    30:
        // 5. ASSERT - Weryfikacja końcowa
        AssertTrue(Condition := Cylinder_RetractHappy.Retracted, 
                   Message := 'Cylinder nie zglosil Retracted po powrocie!');
                   
        TEST_FINISHED();
END_CASE
END_METHOD

END_FUNCTION_BLOCK

// ---- POUs/TESTS/FB_ExecutorNCITable_Test.TcPOU
FUNCTION_BLOCK FB_ExecutorNCITable_Test EXTENDS TcUnit.FB_TestSuite
VAR
    Executor         : FB_Exec_Tangential_FeedTable;
    MockChannel      : FB_MockNciChannelFeedTable;

    Executor_Err     : FB_Exec_Tangential_FeedTable;
    MockChannel_Err  : FB_MockNciChannelFeedTable;

    MockProvider     : FB_MockConfigProvider;
    MockAxisX        : FB_MockAxis;
    MockAxisY        : FB_MockAxis;
    MockAxisZ        : FB_MockAxis;
    RecipeBuilder    : FB_PTPRectangle;
END_VAR

Test_Sequence_ExecutesTableCorrectly();
Test_ChannelError_AbortsSequence();

METHOD Test_ChannelError_AbortsSequence
VAR_INST
    Step : INT := 0;
    TimeoutTimer : TON;
END_VAR
TEST('Test_ChannelError_AbortsSequence');

Executor_Err.CyclicLogic();

TimeoutTimer(IN := (Step > 0 AND Step < 100), PT := T#2S);
IF TimeoutTimer.Q THEN
    AssertTrue(FALSE, 'Timeout! Maszyna stanow utknela.');
    TEST_FINISHED();
    Step := 100;
END_IF

CASE Step OF
    0:
        Executor_Err.RecipeBuilder  := RecipeBuilder;
        Executor_Err.ConfigProvider := MockProvider;
        Executor_Err.AxisX          := MockAxisX;
        Executor_Err.AxisY          := MockAxisY;
        Executor_Err.AxisZ          := MockAxisZ;
        Executor_Err.NciChannel     := MockChannel_Err;

        MockAxisX.MockInPosition := TRUE;
        MockAxisY.MockInPosition := TRUE;
        MockAxisZ.MockInPosition := TRUE;
        MockChannel_Err.MockChannelError := FALSE;

        Executor_Err.Execute();
        Step := 10;

    10:
        IF MockChannel_Err.BuildGroupCallCount > 0 THEN
            MockChannel_Err.MockChannelError := TRUE;
            MockChannel_Err.MockChannelErrorId := 4321;
            Step := 20;
        END_IF

    20:
        IF Executor_Err.Error THEN
            AssertEquals_UDINT(Expected := 4321, 
                               Actual := Executor_Err.ErrorID, 
                               Message := 'Executor nie przepisal ErrorID z kanalu tabelarycznego!');
            TEST_FINISHED();
            Step := 100;
        ELSIF Executor_Err.Done THEN
            AssertTrue(Condition := FALSE, Message := 'Executor zignorowal blad kanalu!');
            TEST_FINISHED();
            Step := 100;
        END_IF
END_CASE
END_METHOD

METHOD Test_Sequence_ExecutesTableCorrectly
VAR_INST
    Step         : INT := 0;
    RecipeConfig : ST_RecipeBuilder_Config;
    TimeoutTimer : TON;
END_VAR
TEST('Test_Sequence_ExecutesTableCorrectly');

Executor.CyclicLogic();

TimeoutTimer(IN := (Step > 0 AND Step < 100), PT := T#2S);
IF TimeoutTimer.Q THEN
    AssertTrue(FALSE, 'Timeout! Maszyna stanow utknela.');
    TEST_FINISHED();
    Step := 100;
END_IF

CASE Step OF
    0:
        RecipeConfig.PanelFrontLength := 1000.0;
        RecipeConfig.PanelFrontWidth  := 1000.0; // <- Wymagane, zeby nie ustawilo 0 sztuk!
        RecipeBuilder.Config := RecipeConfig;
        RecipeBuilder.Build();

        Executor.RecipeBuilder  := RecipeBuilder;
        Executor.ConfigProvider := MockProvider;
        Executor.AxisX          := MockAxisX;
        Executor.AxisY          := MockAxisY;
        Executor.AxisZ          := MockAxisZ;
        Executor.NciChannel     := MockChannel; 

        Step := 10;

    10:
        Executor.Execute();
        Step := 20;

    20:
        IF Executor.Busy THEN
            MockAxisX.MockInPosition := TRUE;
            MockAxisY.MockInPosition := TRUE;
            MockAxisZ.MockInPosition := TRUE;
            Step := 30;
        END_IF

    30:
        IF MockChannel.BuildGroupCallCount > 0 THEN
            MockChannel.MockIsGrouped := TRUE; 
            Step := 40;
        END_IF

    40:
        IF MockChannel.StartFeedTableCallCount > 0 THEN
            MockChannel.MockIsFeedingDone := TRUE;
            Step := 50;
        END_IF

    50:
        IF MockChannel.MockIsFeedingDone THEN
            MockChannel.MockIsChannelDone := TRUE;
            Step := 60;
        END_IF

    60:
        IF MockChannel.UngroupCallCount > 0 THEN
            MockChannel.MockIsGrouped := FALSE;
            Step := 70;
        END_IF

    70:
        IF Executor.Done THEN
            AssertTrue(Condition := TRUE, Message := 'Test OK');
            TEST_FINISHED();
            Step := 100;
        ELSIF Executor.Error THEN
            AssertTrue(Condition := FALSE, Message := 'Wystapil nieoczekiwany Error!');
            TEST_FINISHED();
            Step := 100;
        END_IF
END_CASE
END_METHOD

END_FUNCTION_BLOCK

// ---- POUs/TESTS/Mocks/FB_MockNciChannelFeedTable.TcPOU
FUNCTION_BLOCK FB_MockNciChannelFeedTable EXTENDS FB_ComponentBase IMPLEMENTS I_NciChannel_FeedTable
VAR_INPUT
    MockIsGrouped      : BOOL;
    MockIsReady        : BOOL;
    MockChannelError   : BOOL;
    MockChannelErrorId : UDINT;
    MockIsFeedingDone  : BOOL;
    MockIsChannelDone  : BOOL;
END_VAR
VAR_OUTPUT
    BuildGroupCallCount     : INT;
    StartFeedTableCallCount : INT;
    StopCallCount           : INT;
    UngroupCallCount        : INT;
    ResetCallCount          : INT;
END_VAR

METHOD BuildGroup
BuildGroupCallCount := BuildGroupCallCount + 1;
END_METHOD

PROPERTY ChannelError : BOOL
GET
ChannelError := MockChannelError;
END_GET
END_PROPERTY

PROPERTY ChannelErrorId : UDINT
GET
ChannelErrorId := MockChannelErrorId;
END_GET
END_PROPERTY

PROPERTY IsChannelDone : BOOL
GET
IsChannelDone := MockIsChannelDone;
END_GET
END_PROPERTY

PROPERTY IsFeedingDone : BOOL
GET
IsFeedingDone := MockIsFeedingDone;
END_GET
END_PROPERTY

PROPERTY IsGrouped : BOOL
GET
IsGrouped := MockIsGrouped;
END_GET
END_PROPERTY

PROPERTY IsReady : BOOL
GET
IsReady := MockIsReady;
END_GET
END_PROPERTY

METHOD ResetChannel
ResetCallCount := ResetCallCount + 1;
MockChannelError := FALSE;
MockChannelErrorId := 0;
END_METHOD

METHOD StartFeedTable
VAR_IN_OUT
    stTable : ST_NciFeedGroupTable;
END_VAR
StartFeedTableCallCount := StartFeedTableCallCount + 1;
END_METHOD

METHOD Stop
StopCallCount := StopCallCount + 1;
END_METHOD

METHOD Ungroup
UngroupCallCount := UngroupCallCount + 1;
END_METHOD

END_FUNCTION_BLOCK

// ---- POUs/TESTS/Mocks/FB_MockConfigProvider.TcPOU
FUNCTION_BLOCK FB_MockConfigProvider IMPLEMENTS I_GantryConfigProvider
VAR
    _MockConfig : ST_GantryXYZ_Config;
END_VAR

PROPERTY Config : ST_GantryXYZ_Config
GET
Config := _MockConfig;
END_GET
SET
_MockConfig := Config;
END_SET
END_PROPERTY

END_FUNCTION_BLOCK

// ---- POUs/TESTS/Mocks/FB_MockAxis.TcPOU
FUNCTION_BLOCK FB_MockAxis EXTENDS SPT_Components.FB_Component_BasicAxis
VAR
	_Enabled		: BOOL := FALSE;
	
	_MockVelocity     : LREAL;
    _MockAcceleration : LREAL;
    _MockDeceleration : LREAL;
	
	_ForceError	:	BOOL;
END_VAR

VAR_INPUT
    MockInPosition : BOOL := TRUE;
    MockBusy       : BOOL := FALSE;
END_VAR

PROPERTY Acceleration : LREAL
GET
Acceleration := _MockAcceleration;
END_GET
SET
_MockAcceleration := Acceleration;
END_SET
END_PROPERTY

PROPERTY Busy : BOOL
GET
Busy := MockBusy;
END_GET
END_PROPERTY

METHOD CyclicLogic
SUPER^.CyclicLogic();
END_METHOD

PROPERTY Deceleration : LREAL
GET
Deceleration := _MockDeceleration;
END_GET
SET
_MockDeceleration := Deceleration;
END_SET
END_PROPERTY

METHOD Enable : BOOL
SUPER^.Enable(); 
_Enabled := TRUE;
Enable := TRUE;
END_METHOD

PROPERTY Enabled : BOOL
GET
Enabled := _Enabled;
END_GET
END_PROPERTY

PROPERTY Error : BOOL
GET
Error := _Error;
END_GET
END_PROPERTY

PROPERTY ForceError : BOOL
GET
ForceError := _Error;
END_GET
SET
_Error := ForceError;
END_SET
END_PROPERTY

PROPERTY InPosition : BOOL
GET
InPosition := MockInPosition;
END_GET
END_PROPERTY

METHOD MoveAbsolute : BOOL
VAR_INPUT
	Position	  : LREAL;
	AbortPrevious : BOOL;
END_VAR
MockBusy := FALSE;
MockInPosition := TRUE;
END_METHOD

PROPERTY Velocity : LREAL
GET
Velocity := _MockVelocity;
END_GET
SET
_MockVelocity := Velocity;
END_SET
END_PROPERTY

END_FUNCTION_BLOCK

// ---- POUs/TESTS/FB_ExecutorGCode_Test.TcPOU
FUNCTION_BLOCK FB_ExecutorGCode_Test EXTENDS TcUnit.FB_TestSuite
VAR
    Executor         : FB_Exec_Spindle_GCodeXYZ;
    MockChannel      : FB_MockNciChannel;

    Executor_Err     : FB_Exec_Spindle_GCodeXYZ;
    MockChannel_Err  : FB_MockNciChannel;

    MockProvider     : FB_MockConfigProvider;
    MockAxisX        : FB_MockAxis;
    MockAxisY        : FB_MockAxis;
    MockAxisZ        : FB_MockAxis;
    RecipeBuilder    : FB_PTPRectangle;
END_VAR

Test_Sequence_CallsChannelMethodsCorrectly();
Test_ChannelError_AbortsSequence();

METHOD Test_ChannelError_AbortsSequence
VAR_INST
    Step : INT := 0;
    TimeoutTimer : TON;
END_VAR
TEST('Test_ChannelError_AbortsSequence');

Executor_Err.CyclicLogic();

TimeoutTimer(IN := (Step > 0 AND Step < 100), PT := T#2S);
IF TimeoutTimer.Q THEN
    AssertTrue(FALSE, 'Timeout! Maszyna stanow utknela.');
    TEST_FINISHED();
    Step := 100;
END_IF

CASE Step OF
    0:
        Executor_Err.RecipeBuilder  := RecipeBuilder;
        Executor_Err.ConfigProvider := MockProvider;
        Executor_Err.AxisX          := MockAxisX;
        Executor_Err.AxisY          := MockAxisY;
        Executor_Err.AxisZ          := MockAxisZ;
        Executor_Err.NciChannel     := MockChannel_Err;

        MockAxisX.MockInPosition := TRUE;
        MockAxisY.MockInPosition := TRUE;
        MockAxisZ.MockInPosition := TRUE;
        MockChannel_Err.MockChannelError := FALSE;

        Executor_Err.Execute();
        Step := 10;
        
    10:
        IF MockChannel_Err.BuildGroupCallCount > 0 THEN
            MockChannel_Err.MockChannelError := TRUE;
            MockChannel_Err.MockChannelErrorId := 1234;
            Step := 20;
        END_IF

    20:
        IF Executor_Err.Error THEN
            AssertEquals_UDINT(Expected := 1234, 
                               Actual := Executor_Err.ErrorID, 
                               Message := 'Executor nie przepisal ErrorID z kanalu!');
            TEST_FINISHED();
            Step := 100; 
        ELSIF Executor_Err.Done THEN
            AssertTrue(Condition := FALSE, Message := 'Executor zignorowal blad kanalu!');
            TEST_FINISHED();
            Step := 100; 
        END_IF
END_CASE
END_METHOD

METHOD Test_Sequence_CallsChannelMethodsCorrectly
VAR_INST
    Step         : INT := 0;
    RecipeConfig : ST_RecipeBuilder_Config;
    TimeoutTimer : TON;
END_VAR
TEST('Test_Sequence_CallsChannelMethodsCorrectly');

Executor.CyclicLogic();

TimeoutTimer(IN := (Step > 0 AND Step < 100), PT := T#2S);
IF TimeoutTimer.Q THEN
    AssertTrue(FALSE, 'Timeout! Maszyna stanow utknela.');
    TEST_FINISHED();
    Step := 100;
END_IF

CASE Step OF
    0:
        RecipeConfig.PanelFrontLength := 1000.0;
        RecipeConfig.PanelFrontWidth  := 1000.0; // <- Wymagane, zeby nie ustawilo 0 sztuk!
        RecipeBuilder.Config := RecipeConfig;
        RecipeBuilder.Build();

        Executor.RecipeBuilder  := RecipeBuilder;
        Executor.ConfigProvider := MockProvider;
        Executor.AxisX          := MockAxisX;
        Executor.AxisY          := MockAxisY;
        Executor.AxisZ          := MockAxisZ;
        Executor.NciChannel     := MockChannel;
        Step := 10;

    10:
        Executor.Execute();
        Step := 20;

    20:
        IF Executor.Busy THEN
            MockAxisX.MockInPosition := TRUE;
            MockAxisY.MockInPosition := TRUE;
            MockAxisZ.MockInPosition := TRUE;
            Step := 30;
        END_IF

    30:
        IF MockChannel.BuildGroupCallCount > 0 THEN
            MockChannel.MockIsGrouped := TRUE;
            Step := 40;
        END_IF

    40:
        IF MockChannel.LoadProgramCallCount > 0 THEN
            AssertEquals_STRING(Expected := '', Actual := MockChannel.LoadedProgramPath, Message := 'Zla sciezka przekazana do kanalu!');
            MockChannel.MockIsProgramLoaded := TRUE;
            Step := 50;
        END_IF

    50:
        IF MockChannel.StartCallCount > 0 THEN
            MockChannel.MockIsReady := TRUE;
            Step := 60;
        END_IF

    60:
        IF MockChannel.UngroupCallCount > 0 THEN
            MockChannel.MockIsGrouped := FALSE;
            Step := 70;
        END_IF

    70:
        IF Executor.Done THEN
            AssertTrue(Condition := TRUE, Message := 'Test OK');
            TEST_FINISHED();
            Step := 100;
        ELSIF Executor.Error THEN
            AssertTrue(Condition := FALSE, Message := 'Wystapil Error!');
            TEST_FINISHED();
            Step := 100;
        END_IF
END_CASE
END_METHOD

END_FUNCTION_BLOCK

// ---- POUs/TESTS/Mocks/FB_MockNciChannel.TcPOU
FUNCTION_BLOCK FB_MockNciChannel EXTENDS FB_ComponentBase IMPLEMENTS I_NciChannel_GCode
VAR_INPUT
    MockIsGrouped      : BOOL;
    MockIsProgramLoaded: BOOL;
    MockIsReady        : BOOL;
    MockIsMoving       : BOOL;
    MockChannelError   : BOOL;
    MockChannelErrorId : UDINT;
END_VAR
VAR_OUTPUT
    BuildGroupCallCount : INT;
    LoadProgramCallCount: INT;
    StartCallCount      : INT;
    StopCallCount       : INT;
    UngroupCallCount    : INT;
    ResetCallCount      : INT;
    LoadedProgramPath   : STRING(255);
END_VAR

METHOD BuildGroup
BuildGroupCallCount := BuildGroupCallCount + 1;
END_METHOD

PROPERTY ChannelError : BOOL
GET
ChannelError := MockChannelError;
END_GET
END_PROPERTY

PROPERTY ChannelErrorId : UDINT
GET
ChannelErrorId := MockChannelErrorId;
END_GET
END_PROPERTY

PROPERTY IsGrouped : BOOL
GET
IsGrouped := MockIsGrouped;
END_GET
END_PROPERTY

PROPERTY IsMoving : BOOL
GET
IsMoving := MockIsMoving;
END_GET
END_PROPERTY

PROPERTY IsProgramLoaded : BOOL
GET
IsProgramLoaded := MockIsProgramLoaded;
END_GET
END_PROPERTY

PROPERTY IsReady : BOOL
GET
IsReady := MockIsReady;
END_GET
END_PROPERTY

METHOD LoadProgram
VAR_INPUT
    sProgramPath : STRING(255);
END_VAR
LoadProgramCallCount := LoadProgramCallCount + 1;
LoadedProgramPath := sProgramPath;
END_METHOD

METHOD ResetChannel
ResetCallCount := ResetCallCount + 1;
MockChannelError := FALSE;
MockChannelErrorId := 0;
END_METHOD

METHOD Start
StartCallCount := StartCallCount + 1;
END_METHOD

METHOD Stop
StopCallCount := StopCallCount + 1;
END_METHOD

METHOD Ungroup
UngroupCallCount := UngroupCallCount + 1;
END_METHOD

END_FUNCTION_BLOCK

// ---- POUs/TESTS/FB_FeedBuilderRoundedRect_Test.TcPOU
FUNCTION_BLOCK FB_FeedBuilderRoundedRect_Test EXTENDS TcUnit.FB_TestSuite
VAR
    Builder    : FB_FeedRoundedRectangle;
    MockWriter : FB_MockGeometryWriter;
    Config     : ST_RecipeBuilder_Config;
END_VAR

Test_Calculates_Footprint_And_StartPoint();
Test_Generates_Lines_And_Arcs_With_Radius();
Test_Zero_Radius_Generates_Only_Lines();

METHOD Test_Calculates_Footprint_And_StartPoint
VAR
    WasBuilt : BOOL;
END_VAR
TEST('Test_Calculates_Footprint_And_StartPoint');

// 1. ARRANGE
Config.PanelFrontWidth  := 300.0;
Config.PanelFrontLength := 400.0;
Config.Radius           := 10.0;
Config.CuttingOverpass  := 0.0; // Upraszczamy Footprint
Config.GroovingOverpass := 0.0;

Builder.Config := Config;
Builder.GeometryWriter := MockWriter; // Wstrzykujemy mock

// 2. ACT
WasBuilt := Builder.Build();

// 3. ASSERT
AssertTrue(Condition := WasBuilt, Message := 'Recepta zwrocila FALSE przy probie Build()!');

AssertEquals_REAL(Expected := 300.0, 
                  Actual := Builder.FootprintX, 
                  Delta := 0.01, 
                  Message := 'Zle wyliczony FootprintX dla zaokraglonego prostokata!');

AssertEquals_REAL(Expected := 400.0, 
                  Actual := Builder.FootprintY, 
                  Delta := 0.01, 
                  Message := 'Zle wyliczony FootprintY dla zaokraglonego prostokata!');

// Sprawdzamy czy start w osi X to srodek detalu (zgodnie z kodem TotalX / 2.0)
AssertEquals_LREAL(Expected := 150.0, 
                   Actual := MockWriter.LastStartX, 
                   Delta := 0.01, 
                   Message := 'Punt Startowy NCI X nie znajduje sie na srodku dolnej krawedzi!');

TEST_FINISHED();
END_METHOD

METHOD Test_Generates_Lines_And_Arcs_With_Radius
VAR
    WasBuilt : BOOL;
END_VAR
TEST('Test_Generates_Lines_And_Arcs_With_Radius');

// 1. ARRANGE
Config.PanelFrontWidth  := 200.0;
Config.PanelFrontLength := 300.0;
Config.Radius           := 20.0;
Builder.Config := Config;
Builder.GeometryWriter := MockWriter;

// Uzywamy nowej metody do resetowania mocka
MockWriter.ResetCounters();

// 2. ACT
WasBuilt := Builder.Build();

// 3. ASSERT
// 4 rogi z promieniem > 0 powinny wygenerować 4 łuki
AssertEquals_INT(Expected := 4, 
                 Actual := MockWriter.AddArcCount, 
                 Message := 'Oczekiwano wygenerowania 4 lukow (AddArc)!');

// Dojazd od punktu srodkowego (1), miedzy 4 rogami (3), i powrot do srodka (1) = 5 linii.
AssertEquals_INT(Expected := 5, 
                 Actual := MockWriter.AddLineCount, 
                 Message := 'Oczekiwano wygenerowania 5 linii prostych (AddLine)!');

TEST_FINISHED();
END_METHOD

METHOD Test_Zero_Radius_Generates_Only_Lines
VAR
    WasBuilt : BOOL;
END_VAR
TEST('Test_Zero_Radius_Generates_Only_Lines');

// 1. ARRANGE
Config.PanelFrontWidth  := 200.0;
Config.PanelFrontLength := 300.0;
Config.Radius           := 0.0; // Promień ZERO (ostry prostokąt)
Builder.Config := Config;
Builder.GeometryWriter := MockWriter;

// Uzywamy nowej metody do resetowania mocka
MockWriter.ResetCounters();

// 2. ACT
WasBuilt := Builder.Build();

// 3. ASSERT
// Przy promieniu = 0 kod recepty ma warunek IF Radius > 0, wiec łuki się nie dodadzą
AssertEquals_INT(Expected := 0, 
                 Actual := MockWriter.AddArcCount, 
                 Message := 'Przy promieniu 0 wygenerowano luki!');

AssertEquals_INT(Expected := 5, 
                 Actual := MockWriter.AddLineCount, 
                 Message := 'Oczekiwano wygenerowania 5 linii prostych (prostokat bez zaokraglen)!');

TEST_FINISHED();
END_METHOD

END_FUNCTION_BLOCK

// ---- POUs/TESTS/Mocks/FB_MockGeometryWriter.TcPOU
FUNCTION_BLOCK FB_MockGeometryWriter IMPLEMENTS I_GeometryWriter
VAR_OUTPUT
    ClearCount                     : INT;
    EnableTangentialFollowingCount : INT;
    AddStartPointCount             : INT;
    AddLineCount                   : INT;
    AddArcCount                    : INT;
    EndTableCount                  : INT;
    
    // Ostatnie parametry ze StartPoint (do weryfikacji)
    LastStartX : LREAL;
    LastStartY : LREAL;
END_VAR

METHOD AddArc : BOOL
VAR_INPUT
    TargetX    : LREAL;
    TargetY    : LREAL;
    CenterX    : LREAL;
    CenterY    : LREAL;
    Velo       : LREAL;
    Clockwise  : BOOL;
END_VAR
AddArcCount := AddArcCount + 1;
AddArc := TRUE;
END_METHOD

METHOD AddLine : BOOL
VAR_INPUT
    TargetX : LREAL;
    TargetY : LREAL;
    Velo    : LREAL;
END_VAR
AddLineCount := AddLineCount + 1;
AddLine := TRUE;
END_METHOD

METHOD AddStartPoint : BOOL
VAR_INPUT
    TargetX : LREAL;
    TargetY : LREAL;
END_VAR
AddStartPointCount := AddStartPointCount + 1;
LastStartX := TargetX;
LastStartY := TargetY;
AddStartPoint := TRUE;
END_METHOD

METHOD Clear : BOOL
VAR_INPUT
END_VAR
ClearCount := ClearCount + 1;
Clear := TRUE;
END_METHOD

METHOD EnableTangentialFollowing : BOOL
VAR_INPUT
END_VAR
EnableTangentialFollowingCount := EnableTangentialFollowingCount + 1;
EnableTangentialFollowing := TRUE;
END_METHOD

METHOD EndTable : BOOL
VAR_INPUT
END_VAR
EndTableCount := EndTableCount + 1;
EndTable := TRUE;
END_METHOD

METHOD ResetCounters
ClearCount := 0;
EnableTangentialFollowingCount := 0;
AddStartPointCount := 0;
AddLineCount := 0;
AddArcCount := 0;
EndTableCount := 0;
LastStartX := 0.0;
LastStartY := 0.0;
END_METHOD

END_FUNCTION_BLOCK

// ---- POUs/TESTS/FB_NciChannelTangential_Test.TcPOU
FUNCTION_BLOCK FB_NciChannelTangential_Test EXTENDS TcUnit.FB_TestSuite
VAR
    ChannelTan  : FB_NciChannelTangential;
    DummyTable  : ST_NciFeedGroupTable;
END_VAR

Test_StartFeedTable_ResetsDoneFlags();
Test_ResetChannel_ClearsErrors();
Test_BuildExtGroup_ClearsGroupedFlag();

METHOD Test_BuildExtGroup_ClearsGroupedFlag
VAR_INST
END_VAR
TEST('Test_BuildExtGroup_ClearsGroupedFlag');

// ACT - Budowanie grupy zawierającej dodatkowo oś Q1
ChannelTan.BuildGroup();

// ASSERT
AssertFalse(Condition := ChannelTan.IsGrouped,
            Message := 'IsGrouped nie zostalo zresetowane przy wywolaniu BuildGroup na EXT grupie!');
AssertFalse(Condition := ChannelTan.ChannelError,
            Message := 'Bledy kanalu tangencjalnego nie zostaly zresetowane przy probie BuildGroup!');

TEST_FINISHED();
END_METHOD

METHOD Test_ResetChannel_ClearsErrors
VAR_INST
END_VAR
TEST('Test_ResetChannel_ClearsErrors');

// ACT
ChannelTan.ResetChannel();

// ASSERT
AssertFalse(Condition := ChannelTan.ChannelError,
            Message := 'Flaga bledu kanalu tangencjalnego nie zniknela po wywolaniu ResetChannel!');
AssertEquals_UDINT(Expected := 0, 
                   Actual := ChannelTan.ChannelErrorId, 
                   Message := 'ID bledu nie zostalo wyzerowane w kanale tangencjalnym!');

TEST_FINISHED();
END_METHOD

METHOD Test_StartFeedTable_ResetsDoneFlags
VAR_INST
END_VAR
TEST('Test_StartFeedTable_ResetsDoneFlags');

// ACT - Przekazujemy strukturę z tabelą i startujemy feedowanie punktów
ChannelTan.StartFeedTable(stTable := DummyTable);

// ASSERT - Flagi końca powinny być natychmiast wyzerowane
AssertFalse(Condition := ChannelTan.IsFeedingDone,
            Message := 'IsFeedingDone powinno byc FALSE na starcie interpolacji tabelarycznej!');
AssertFalse(Condition := ChannelTan.IsChannelDone,
            Message := 'IsChannelDone powinno byc FALSE na starcie interpolacji tabelarycznej!');

TEST_FINISHED();
END_METHOD

END_FUNCTION_BLOCK

// ---- POUs/TESTS/FB_NciChannel_Test.TcPOU
FUNCTION_BLOCK FB_NciChannel_Test EXTENDS TcUnit.FB_TestSuite
VAR
    Channel : FB_NciChannel;
END_VAR

Test_LoadProgram_ClearsLoadedFlag();
Test_ResetChannel_ClearsErrors();
Test_BuildGroup_ClearsGroupedFlag();
Test_Real_BuildGroup_Integration();
Test_DisconnectedState_ReturnsNotReady();

METHOD Test_BuildGroup_ClearsGroupedFlag
VAR_INST
    Executed : BOOL;
END_VAR
TEST('Test_BuildGroup_ClearsGroupedFlag');
IF NOT Executed THEN
    Channel.BuildGroup();
    AssertFalse(Condition := Channel.IsGrouped, Message := 'IsGrouped nie zostalo zresetowane przy wywolaniu BuildGroup!');
    AssertFalse(Condition := Channel.ChannelError, Message := 'Bledy kanalu nie zostaly zresetowane przy probie BuildGroup!');
    TEST_FINISHED();
    Executed := TRUE;
END_IF
END_METHOD

METHOD Test_DisconnectedState_ReturnsNotReady
VAR_INST
    Executed : BOOL;
END_VAR
TEST('Test_DisconnectedState_ReturnsNotReady');
IF NOT Executed THEN
    AssertFalse(Condition := Channel.IsReady, Message := 'IsReady zwrocilo TRUE pomimo braku fizycznego polaczenia z NC!');
    AssertFalse(Condition := Channel.IsMoving, Message := 'IsMoving zwrocilo TRUE pomimo braku fizycznego polaczenia z NC!');
    TEST_FINISHED();
    Executed := TRUE;
END_IF
END_METHOD

METHOD Test_LoadProgram_ClearsLoadedFlag
VAR_INST
    Executed : BOOL;
END_VAR
TEST('Test_LoadProgram_ClearsLoadedFlag');
IF NOT Executed THEN
    Channel.LoadProgram('C:\test_path.nc');
    AssertFalse(Condition := Channel.IsProgramLoaded, Message := 'Flaga IsProgramLoaded nie zostala zresetowana!');
    TEST_FINISHED();
    Executed := TRUE;
END_IF
END_METHOD

METHOD Test_Real_BuildGroup_Integration
VAR_INST
    Step : INT := 0;
    TimeoutTimer : TON;
END_VAR
TEST('Test_Real_BuildGroup_Integration');

// Wstrzykujemy ID osi testowych (odczytane z Twojego tsproj) oraz poprawne ID grupy
Channel.stAxisIds.nX := 5; 
Channel.stAxisIds.nY := 6;
Channel.stAxisIds.nZ := 7;
Channel.nGroupId := 11; // Wirtualna grupa NCI dla testow to 11

Channel.CyclicLogic();

CASE Step OF
    0:
        Channel.BuildGroup();
        Step := 10;

    10:
        TimeoutTimer(IN := TRUE, PT := T#3S);
        
        IF Channel.IsGrouped THEN
            Step := 20;
        ELSIF Channel.ChannelError THEN
            AssertTrue(Condition := FALSE, Message := CONCAT('NC zwrocilo blad! ErrorID: ', UDINT_TO_STRING(Channel.ChannelErrorId)));
            TEST_FINISHED();
        ELSIF TimeoutTimer.Q THEN
            AssertTrue(Condition := FALSE, Message := 'Timeout! NC nie odpowiedzialo.');
            TEST_FINISHED();
        END_IF

    20:
        AssertTrue(Condition := Channel.IsGrouped, Message := 'Grupa powinna byc zgloszona jako gotowa!');
        Channel.Ungroup();
        Step := 30;

    30:
        IF NOT Channel.IsGrouped THEN
            TimeoutTimer(IN := FALSE);
            TEST_FINISHED();
            Step := 100;
        END_IF
END_CASE
END_METHOD

METHOD Test_ResetChannel_ClearsErrors
VAR_INST
    Executed : BOOL;
END_VAR
TEST('Test_ResetChannel_ClearsErrors');
IF NOT Executed THEN
    Channel.ResetChannel();
    AssertFalse(Condition := Channel.ChannelError, Message := 'Flaga bledu kanalu nie zniknela po wywolaniu ResetChannel!');
    AssertEquals_UDINT(Expected := 0, Actual := Channel.ChannelErrorId, Message := 'ID bledu nie zostalo wyzerowane!');
    TEST_FINISHED();
    Executed := TRUE;
END_IF
END_METHOD

END_FUNCTION_BLOCK

// ---- POUs/TESTS/FB_GantryXYZ_Test.TcPOU
FUNCTION_BLOCK FB_GantryXYZ_Test EXTENDS TcUnit.FB_TestSuite
VAR
	Gantry : FB_GantryXYZ;
END_VAR

Test_ApplyProfile_Applies_Correct_Dynamics();
Test_Speeds_Never_Zero_Or_Negative();
//Test_StateChanged_Updates_Profile(); //Needs to be investigated

METHOD Test_ApplyProfile_Applies_Correct_Dynamics
VAR_INPUT
END_VAR
TEST('Test_ApplyProfile_Applies_Correct_Dynamics');

// 1. ACT - Aplikujemy profil Homing (powolny, otwarte limity)
Gantry.ApplyProfile(E_MachineProfile.eHoming);

// 2. ASSERT - Akceleracja osi X powinna wynosić 200.0
AssertEquals_LREAL(Expected := 200.0, 
                   Actual := Gantry.RefAxisX.Acceleration, 
                   Delta := 0.01, 
                   Message := 'ApplyProfile: Blad akceleracji X dla profilu Homing');

// 3. ACT - Aplikujemy profil Production (agresywny)
Gantry.ApplyProfile(E_MachineProfile.eProduction);

// 4. ASSERT - Akceleracja osi X powinna wynosić 1500.0
AssertEquals_LREAL(Expected := 1500.0, 
                   Actual := Gantry.RefAxisX.Acceleration, 
                   Delta := 0.01, 
                   Message := 'ApplyProfile: Blad akceleracji X dla profilu Production');

// 5. ACT - Aplikujemy profil Manual (pośredni)
Gantry.ApplyProfile(E_MachineProfile.eManual);

// 6. ASSERT - Akceleracja osi X powinna wynosić 500.0
AssertEquals_LREAL(Expected := 500.0, 
                   Actual := Gantry.RefAxisX.Acceleration, 
                   Delta := 0.01, 
                   Message := 'ApplyProfile: Blad akceleracji X dla profilu Manual');

TEST_FINISHED();
END_METHOD

METHOD Test_Speeds_Never_Zero_Or_Negative
VAR
    BadConfig    : ST_GantryXYZ_Config;
    ActualConfig : ST_GantryXYZ_Config;
END_VAR
TEST('Test_Speeds_Never_Zero_Or_Negative');

// 1. ARRANGE - Złe dane (np. wpisane przez uszkodzone HMI lub błąd ludzki)
BadConfig.RapidSpeedX := 0.0;        // Zero! Oś nigdy nie dojedzie, zawiesi maszynę stanów
BadConfig.CuttingSpeedXY := -50.0;    // Ujemna prędkość!
BadConfig.GroovingSpeedZ := -0.01;   // Prędkość zagłębiania bliska 0/ujemna
BadConfig.CuttingIdleTime := -2.0;   // Ujemny czas postoju? Timer zwariuje

// 2. ACT - Próba wstrzyknięcia do Gantry
Gantry.Config := BadConfig;
ActualConfig := Gantry.Config; // Odczytujemy stan po "obronie" przez Set

// 3. ASSERT - Sprawdzamy czy Gantry ustawiło bezpieczne minima
AssertEquals_REAL(Expected := 1.0, 
                  Actual := ActualConfig.RapidSpeedX, 
                  Delta := 0.01, 
                  Message := 'RapidSpeedX rowne 0 zostalo przepuszczone!');

AssertEquals_REAL(Expected := 1.0, 
                  Actual := ActualConfig.CuttingSpeedXY, 
                  Delta := 0.01, 
                  Message := 'Ujemna predkosc ciecia przeszla do systemu!');

AssertEquals_REAL(Expected := 1.0, 
                  Actual := ActualConfig.GroovingSpeedZ, 
                  Delta := 0.01, 
                  Message := 'Ujemna/Zerowa predkosc zaglabiania (Z) przeszla!');
                  
AssertEquals_REAL(Expected := 0.0, 
                  Actual := ActualConfig.CuttingIdleTime, 
                  Delta := 0.01, 
                  Message := 'Ujemny czas oczekiwania przeszedl do systemu!');

TEST_FINISHED();
END_METHOD

METHOD Test_StateChanged_Updates_Profile
VAR_INST
    Step : INT := 0;
    Watchdog : TON; // Zabezpieczenie przed zawieszeniem IDE
END_VAR
TEST('Test_StateChanged_Updates_Profile');

// Krytyczne: Wywołujemy logikę Gantry raz na cykl PLC, BEZ ŻADNYCH PĘTLI WHILE/FOR!
Gantry.CyclicLogic();

// Zabezpieczenie testu: jeżeli maszyna PackML utknie i nie zmieni stanu,
// po 2 sekundach przerywamy test, by chronić IDE przed zawieszeniem.
Watchdog(IN := (Step > 0 AND Step < 100), PT := T#2S);
IF Watchdog.Q THEN
    AssertTrue(Condition := FALSE, Message := 'Timeout testu - PackML utknelo w jednym ze stanow! Prawdopodobnie odrzucono komende.');
    TEST_FINISHED();
    Step := 100; // Blokada przed dalszym wykonywaniem
END_IF

CASE Step OF
    0:
        // 1. Zmieniamy tryb na Manualny (od razu na starcie)
        Gantry.ChangeMode(E_PMLUnitMode.ePMLUnitMode_Manual);
        Step := 5;

    5:
        // Czekamy aż PackML fizycznie "zrozumie" zmianę trybu
        IF Gantry.CurrentMode = E_PMLUnitMode.ePMLUnitMode_Manual THEN
            // Zrzucamy maszynę do bezpiecznego stanu Aborted
            Gantry.ChangeState(E_PMLCommand.ePMLCommand_Abort);
            Step := 10;
        END_IF

    10:
        // Czekamy na wejście w Aborted
        IF Gantry.CurrentState = E_PMLState.ePMLState_Aborted THEN
            
            // W trybie Manual zawsze profil ma być ustawiony na Acc=500.0
            AssertEquals_LREAL(Expected := 500.0, 
                               Actual := Gantry.RefAxisX.Acceleration, 
                               Delta := 0.01, 
                               Message := 'Tryb Manualny nie zaladowal prawidlowego profilu!');

            // Zmieniamy tryb z powrotem na produkcyjny
            Gantry.ChangeMode(E_PMLUnitMode.ePMLUnitMode_Production);
            Step := 15;
        END_IF

    15:
        // Czekamy aż PackML potwierdzi tryb produkcyjny
        IF Gantry.CurrentMode = E_PMLUnitMode.ePMLUnitMode_Production THEN
            // Ze stanu Aborted przechodzimy komendą Clear
            Gantry.ChangeState(E_PMLCommand.ePMLCommand_Clear);
            Step := 20;
        END_IF
        
    20:
        // Maszyna po "Clearing" wejdzie w stan "Stopped"
        IF Gantry.CurrentState = E_PMLState.ePMLState_Stopped THEN
            
            // DOPIERO stąd można bezpiecznie wezwać komendę Reset!
            Gantry.ChangeState(E_PMLCommand.ePMLCommand_Reset);
            Step := 30;
        END_IF

    30:
        // Łapiemy moment wejścia w Resetting
        IF Gantry.CurrentState = E_PMLState.ePMLState_Resetting THEN
            
            // To nasz ostateczny sprawdzian: StateChanged() powinno było podmienić profil!
            AssertEquals_LREAL(Expected := 200.0, 
                               Actual := Gantry.RefAxisX.Acceleration, 
                               Delta := 0.01, 
                               Message := 'Rozpoczecie bazowania (Resetting) nie zmienilo profilu maszyny na Homing!');
                               
            TEST_FINISHED(); // Sukces!
            Step := 100; // Koniec
        END_IF
END_CASE
END_METHOD

END_FUNCTION_BLOCK

// ---- POUs/TESTS/FB_ExecutorCut_Test.TcPOU
FUNCTION_BLOCK FB_ExecutorCut_Test EXTENDS TcUnit.FB_TestSuite 
VAR
    Executor : FB_Exec_Pneumatic_PTP;
	Executor_Unhappy     : FB_Exec_Pneumatic_PTP;
	
	MockConfigProvider : FB_MockConfigProvider;

    MockCylinder : FB_MockCylinder;
	MockCylinder_Unhappy : FB_MockCylinder;
    MockAxisX    : FB_MockAxis := (Name := 'MockX');
    MockAxisY    : FB_MockAxis := (Name := 'MockY');
    MockAxisZ    : FB_MockAxis := (Name := 'MockZ');
    
    TestRecipe   : FB_PTPBorgoWings;

	
	Executor_Zero       : FB_Exec_Pneumatic_PTP;
    MockCylinder_Zero   : FB_MockCylinder;
    BuilderArona        : FB_PTPArona; // Arona to nasza wydmuszka, zwraca 0 segmentów!

    Executor_AxisErr    : FB_Exec_Pneumatic_PTP;
    MockAxisX_Err       : FB_MockAxis;

    Executor_CutY       : FB_Exec_Pneumatic_PTP;
    MockCylinder_CutY   : FB_MockCylinder;
	
	Executor_Nesting : FB_Exec_Pneumatic_PTP;
    MockCylinder_Nesting : FB_MockCylinder;
	
END_VAR

Test_AxisError_AbortsSequence();
Test_Executes_CutY_Direction();
Test_Executes_Nesting_Copies();
Test_Sequence_AbortsOnCylinderError();
Test_Sequence_ExecutesCutsCorrectly();
Test_ZeroSegments_FinishesImmediately();

METHOD Test_AxisError_AbortsSequence
VAR_INST
    i : INT;
    RecipeConfig : ST_RecipeBuilder_Config; 
END_VAR


TEST('Test_AxisError_AbortsSequence');

// 1. ARRANGE - Używamy poprawnej receptury (BorgoWings)
RecipeConfig.PanelFrontLength := 1000.0;  
TestRecipe.Config := RecipeConfig;        
TestRecipe.Build();                       
Executor_AxisErr.RecipeBuilder  := TestRecipe; 
Executor_AxisErr.ConfigProvider := MockConfigProvider; // Poprawiona nazwa
Executor_AxisErr.Cylinder       := MockCylinder;
Executor_AxisErr.AxisX          := MockAxisX_Err; // Podpinamy złośliwą oś
Executor_AxisErr.AxisY          := MockAxisY;
Executor_AxisErr.AxisZ          := MockAxisZ;
Executor_AxisErr.CutDirection   := E_CutDirection.eCutX;

MockAxisX_Err.ForceError := TRUE; // Zmuszamy oś do błędu!

// 2. ACT
Executor_AxisErr.Execute();

// Puszczamy maszynę stanów. Wpadnie do kroku 10 (dojazd), potem 20 i od razu zobaczy błąd osi (skok do 999).
FOR i := 1 TO 10 DO
    Executor_AxisErr.CyclicLogic();
END_FOR

// 3. ASSERT
AssertTrue(Condition := Executor_AxisErr.Error, 
           Message := 'Executor nie zglosil bledu, gdy os ulegla awarii!');

AssertFalse(Condition := Executor_AxisErr.Done, 
            Message := 'Executor zglosil sukces (Done), pomimo bledu osi!');

TEST_FINISHED();
END_METHOD

METHOD Test_Executes_CutY_Direction
VAR_INST
    Step : INT := 0;
    RecipeConfig : ST_RecipeBuilder_Config;
END_VAR
TEST('Test_Executes_CutY_Direction');

Executor_CutY.CyclicLogic();

CASE Step OF
    0:
        // 1. ARRANGE - Receptura BorgoWings ma dokładnie 6 cięć Y
        RecipeConfig.PanelFrontLength := 1000.0;
        TestRecipe.Config := RecipeConfig;
        TestRecipe.Build(); 
        
        Executor_CutY.RecipeBuilder  := TestRecipe;
		Executor_CutY.ConfigProvider := MockConfigProvider;
        Executor_CutY.Cylinder       := MockCylinder_CutY;
        Executor_CutY.AxisX          := MockAxisX;
        Executor_CutY.AxisY          := MockAxisY;
        Executor_CutY.AxisZ          := MockAxisZ;
        
        // Ustawiamy cięcie wzdłuż osi Y!
        Executor_CutY.CutDirection   := E_CutDirection.eCutY; 
        
        Step := 10;
        
    10:
        // 2. ACT
        Executor_CutY.Execute();
        Step := 20;
        
    20:
        // Czekamy na koniec asynchronicznej sekwencji
        IF Executor_CutY.Done THEN
            Step := 30;
        ELSIF Executor_CutY.Error THEN
            AssertTrue(FALSE, 'Wyrzucono blad podczas ciecia Y!');
            TEST_FINISHED();
        END_IF
        
    30:
        // 3. ASSERT - Weryfikujemy ilość cięć (BorgoWings = 6)
        AssertEquals_INT(Expected := 6, 
                         Actual := MockCylinder_CutY.ExtendCallCount, 
                         Message := 'Zla liczba wysuniec cylindra przy cieciu Y!');
                         
        TEST_FINISHED();
END_CASE
END_METHOD

METHOD Test_Executes_Nesting_Copies
VAR_INST
    Step         : INT := 0;
    RecipeConfig : ST_RecipeBuilder_Config;
    TestConfig   : ST_GantryXYZ_Config;
    

    LocalTestRecipe : FB_PTPBorgoWings;
    LocalConfigProvider : FB_MockConfigProvider;
END_VAR
TEST('Test_Executes_Nesting_Copies');
Executor_Nesting.CyclicLogic(); 

CASE Step OF
    0:
        // 1. ARRANGE
        // Wykorzystujemy BorgoWings, które domyślnie posiada 6 segmentów CutX
        RecipeConfig.PanelFrontLength := 300.0;
        RecipeConfig.PanelHeight := 100.0;
        RecipeConfig.PanelFrontWidth := 300.0;
        
        // Wymuszamy 2 kopie w X i 2 kopie w Y
        RecipeConfig.FillAll := FALSE;
        RecipeConfig.RequestedCopiesX := 2;
        RecipeConfig.RequestedCopiesY := 2;
        
        LocalTestRecipe.Config := RecipeConfig;
        LocalTestRecipe.Build(); 
        
        TestConfig.CuttingSpeedXY := 100;
        TestConfig.RapidSpeedX := 100;
        TestConfig.CuttingIdleTime := 0.0;
        // Szybki test
        
        // Podpinamy wyizolowane zależności
        LocalConfigProvider.Config := TestConfig;
        Executor_Nesting.RecipeBuilder  := LocalTestRecipe;
        Executor_Nesting.ConfigProvider := LocalConfigProvider;
        Executor_Nesting.Cylinder       := MockCylinder_Nesting;
        Executor_Nesting.AxisX          := MockAxisX;
        Executor_Nesting.AxisY          := MockAxisY;
        Executor_Nesting.AxisZ          := MockAxisZ;
        Executor_Nesting.CutDirection   := E_CutDirection.eCutX; 
        
        Step := 10;
        
    10:
        // 2. ACT
        Executor_Nesting.Execute();
        Step := 20;
        
    20:
        IF Executor_Nesting.Done THEN
            Step := 30;
        ELSIF Executor_Nesting.Error THEN
            AssertTrue(FALSE, 'Executor zwrocil Error zamiast Done przy Nestingu!');
            TEST_FINISHED();
        END_IF
        
    30:
        // 3. ASSERT
        // BorgoWings ma 6 cięć X na jedną sztukę.
        // 2 kopie X * 2 kopie Y = 4 sztuki.
        // 4 sztuki * 6 cięć = 24 wysunięcia siłownika!
        AssertEquals_INT(Expected := 24, 
                         Actual := MockCylinder_Nesting.ExtendCallCount, 
                         Message := 'Zla liczba ciec przy multiplexowaniu (Nestingu)!');
        TEST_FINISHED();
END_CASE
END_METHOD

METHOD Test_Sequence_AbortsOnCylinderError
VAR_INST
    Step : INT := 0;
    RecipeConfig : ST_RecipeBuilder_Config;
	TestConfig : ST_GantryXYZ_Config;
END_VAR


TEST('Test_Sequence_AbortsOnCylinderError');

Executor_Unhappy.CyclicLogic();

CASE Step OF
    0:
        // 1. ARRANGE - Przygotowanie receptury BorgoWings (6 cięć)
        RecipeConfig.PanelFrontLength := 1000.0;
        TestRecipe.Config := RecipeConfig;
        TestRecipe.Build(); 
		
		TestConfig.CuttingSpeedXY := 10;    
		TestConfig.GroovingSpeedXY := 10;
		TestConfig.RapidSpeedX := 10;
		TestConfig.RapidSpeedY := 10;
	
        
        TestConfig.CuttingIdleTime := 0.0; 
        
        // ZMUSZAMY MOCK DO AWARII PRZY 3. PRÓBIE WYSUNIĘCIA
        MockCylinder_Unhappy.FailOnExtendCount := 3;
        
        // Wstrzykujemy zależności do Executora "Unhappy"
		MockConfigProvider.Config := TestConfig; 
		Executor_Unhappy.RecipeBuilder  := TestRecipe;
		Executor_Unhappy.ConfigProvider := MockConfigProvider; 
        Executor_Unhappy.Cylinder       := MockCylinder_Unhappy;
        Executor_Unhappy.AxisX          := MockAxisX;
        Executor_Unhappy.AxisY          := MockAxisY;
        Executor_Unhappy.AxisZ          := MockAxisZ;
        
        Step := 10;
        
    10:
        // 2. ACT - Start maszyny
        Executor_Unhappy.Execute();
        Step := 20;
        
    20:
        // 3. ASSERT - Oczekujemy BŁĘDU, a nie zakończenia sukcesem!
        IF Executor_Unhappy.Error THEN
            Step := 30; // Sukces testu - Executor wyrzucił błąd
        ELSIF Executor_Unhappy.Done THEN
            AssertTrue(FALSE, 'Cylinder zglosil blad, a Executor zignorowal to i zakonczyl sukcesem!');
            TEST_FINISHED();
        END_IF
        
    30:
        // 4. ASSERT - Weryfikacja dokładnego zachowania podczas awarii
        
        // Oczekujemy, że wysunięcie zostało wywołane dokładnie 3 razy i ani razu więcej
        AssertEquals_INT(Expected := 3, 
                         Actual := MockCylinder_Unhappy.ExtendCallCount, 
                         Message := 'Executor nie zatrzymal sie po bledzie na 3. cieciu!');
                         
        // Oczekujemy, że wsunięcie zostało wywołane tylko 2 razy 
        // (bo przy trzecim wysunięciu był błąd, więc sekwencja spadła z rowerka przed chowaniem!)
        AssertEquals_INT(Expected := 2, 
                         Actual := MockCylinder_Unhappy.RetractCallCount, 
                         Message := 'Bledna liczba wsuniec przed awaria!');
                         
        TEST_FINISHED();
END_CASE
END_METHOD

METHOD Test_Sequence_ExecutesCutsCorrectly
VAR_INST
    Step : INT := 0;
    RecipeConfig : ST_RecipeBuilder_Config;
	TestConfig : ST_GantryXYZ_Config;
END_VAR
TEST('Test_Sequence_ExecutesCutsCorrectly');

// Wywołujemy CyclicLogic dla Executora (Mocki nie potrzebują, bo nic w nich w tle nie tyka)
Executor.CyclicLogic();

CASE Step OF
    0:
        // 1. ARRANGE - Przygotowanie receptury Arona (ma 2 cięcia X)
        RecipeConfig.PanelFrontLength := 1000.0;
        TestRecipe.Config := RecipeConfig;
        TestRecipe.Build(); 
		TestConfig.CuttingSpeedXY := 10;
		TestConfig.GroovingSpeedXY := 10;
		TestConfig.RapidSpeedX := 10;
		TestConfig.RapidSpeedY := 10;
	

        // Czas stabilizacji dla testu ucinamy do zera
        TestConfig.CuttingIdleTime := 0.0; 
        
        // 2. DEPENDENCY INJECTION - Wstrzykujemy nasze Zaślepki!
		MockConfigProvider.Config := TestConfig; 
		Executor.RecipeBuilder  := TestRecipe;
		Executor.ConfigProvider := MockConfigProvider;
        Executor.Cylinder       := MockCylinder;
        Executor.AxisX          := MockAxisX;
        Executor.AxisY          := MockAxisY;
        Executor.AxisZ          := MockAxisZ;
        
        Step := 10;
        
    10:
        // 3. ACT - Start maszyny
        Executor.Execute();
        Step := 20;
        
    20:
        // 4. Czekamy na koniec sekwencji (dzięki mockom to potrwa ułamki sekund)
        IF Executor.Done THEN
            Step := 30;
        ELSIF Executor.Error THEN
            AssertTrue(FALSE, 'Executor zwrocil Error zamiast Done!');
            TEST_FINISHED();
        END_IF
        
    30:
        // 5. ASSERT - Testujemy Logikę Executora szpiegując Siłownik
        // Arona ma 2 cięcia, więc siłownik musi zostać użyty 2 razy
        AssertEquals_INT(Expected := 6, 
                         Actual := MockCylinder.ExtendCallCount, 
                         Message := 'Bledna liczba wysuniec ostrza!');
                         
        AssertEquals_INT(Expected := 6, 
                         Actual := MockCylinder.RetractCallCount, 
                         Message := 'Bledna liczba wsuniec ostrza!');
                         
        TEST_FINISHED();
END_CASE
END_METHOD

METHOD Test_ZeroSegments_FinishesImmediately
VAR_INST
    i : INT;
END_VAR


TEST('Test_ZeroSegments_FinishesImmediately');

// 1. ARRANGE - Arona aktualnie zwraca 0 segmentów (wydmuszka)
Executor_Zero.RecipeBuilder  := BuilderArona;
Executor_Zero.ConfigProvider := MockConfigProvider; 
Executor_Zero.Cylinder       := MockCylinder_Zero;
Executor_Zero.AxisX          := MockAxisX;
Executor_Zero.AxisY          := MockAxisY;
Executor_Zero.AxisZ          := MockAxisZ;
Executor_Zero.CutDirection   := E_CutDirection.eCutX;

// 2. ACT
Executor_Zero.Execute();

// Maszyna stanów potrzebuje dokładnie 3 cykli, aby z kroku 0 wejść w 5, potem w 1000 i zakończyć.
// Puszczamy pętlę na wszelki wypadek np. 5 razy.
FOR i := 1 TO 5 DO
    Executor_Zero.CyclicLogic();
END_FOR

// 3. ASSERT
AssertTrue(Condition := Executor_Zero.Done, 
           Message := 'Executor nie zwrocil Done przy 0 segmentow!');
           
AssertEquals_INT(Expected := 0, 
                 Actual := MockCylinder_Zero.ExtendCallCount, 
                 Message := 'Silownik zostal uruchomiony, chociaz nie bylo ciec!');

TEST_FINISHED();
END_METHOD

END_FUNCTION_BLOCK

// ---- POUs/TESTS/Mocks/FB_MockCylinder.TcPOU
FUNCTION_BLOCK FB_MockCylinder IMPLEMENTS I_Cylinder
VAR
    _Extended  : BOOL;
    _Retracted : BOOL := TRUE;
    
    ExtendCallCount  : INT := 0;
    RetractCallCount : INT := 0;
	

    _Error            : BOOL := FALSE;
END_VAR

VAR_INPUT
	FailOnExtendCount : INT := 0; 
END_VAR

PROPERTY Error : BOOL
GET
Error := _Error;
END_GET
END_PROPERTY

METHOD Extend
ExtendCallCount := ExtendCallCount + 1;

// Symulacja awarii, jeśli dotarliśmy do wyznaczonego limitu
IF FailOnExtendCount > 0 AND ExtendCallCount = FailOnExtendCount THEN
    _Error := TRUE;
    _Extended := FALSE;
ELSE
    _Extended := TRUE;
    _Retracted := FALSE;
END_IF
END_METHOD

PROPERTY Extended : BOOL
GET
Extended := _Extended;
END_GET
END_PROPERTY

METHOD Retract
_Extended := FALSE; 
_Retracted := TRUE; 
RetractCallCount := RetractCallCount + 1;
END_METHOD

PROPERTY Retracted : BOOL
GET
Retracted := _Retracted;
END_GET
END_PROPERTY

END_FUNCTION_BLOCK

// ---- POUs/TESTS/FB_ExecutorGrooveXY_Test.TcPOU
FUNCTION_BLOCK FB_ExecutorGrooveXY_Test EXTENDS TcUnit.FB_TestSuite 
VAR
    // Instancje naszych obiektów testowanych (SUT - System Under Test)
    Executor         : FB_Exec_Spindle_PTP;
    Executor_Zero    : FB_Exec_Spindle_PTP;
    Executor_Unhappy : FB_Exec_Spindle_PTP;

    // Zaślepka konfiguracji
    MockConfigProvider : FB_MockConfigProvider;

    // Zaślepki osi
    MockAxisX     : FB_MockAxis := (Name := 'MockX');
    MockAxisY     : FB_MockAxis := (Name := 'MockY');
    MockAxisZ     : FB_MockAxis := (Name := 'MockZ');
    MockAxisZ_Err : FB_MockAxis := (Name := 'MockZ_Err'); // Złośliwa oś Z
    
    // Budowniczowie receptur
    TestRecipe   : FB_PTPBorgoWings; // Posiada 4 frezowania
    BuilderArona : FB_PTPArona;      // Wydmuszka, posiada 0 frezowań
END_VAR

Test_AxisError_AbortsSequence();
Test_Sequence_ExecutesGroovesCorrectly();
Test_ZeroSegments_FinishesImmediately();

METHOD Test_AxisError_AbortsSequence
VAR_INST
    i : INT;
    RecipeConfig : ST_RecipeBuilder_Config;
    TestConfig   : ST_GantryXYZ_Config;
END_VAR
TEST('Test_AxisError_AbortsSequence');

// 1. ARRANGE - Używamy poprawnej receptury (BorgoWings - 4 frezowania)
RecipeConfig.PanelFrontLength := 1000.0;  
TestRecipe.Config := RecipeConfig;        
TestRecipe.Build();                       

MockConfigProvider.Config := TestConfig;

Executor_Unhappy.RecipeBuilder  := TestRecipe;
Executor_Unhappy.ConfigProvider := MockConfigProvider;
Executor_Unhappy.AxisX          := MockAxisX;
Executor_Unhappy.AxisY          := MockAxisY;
Executor_Unhappy.AxisZ          := MockAxisZ_Err; // Podpinamy złośliwą oś Z

// Zmuszamy oś Z do błędu!
MockAxisZ_Err.ForceError := TRUE;

// 2. ACT
Executor_Unhappy.Execute();

// Puszczamy maszynę stanów (wpadnie w krok dojazdu i powinna wejść w 999)
FOR i := 1 TO 10 DO
    Executor_Unhappy.CyclicLogic();
END_FOR

// 3. ASSERT
AssertTrue(Condition := Executor_Unhappy.Error, 
           Message := 'Executor nie zglosil bledu, gdy os Z ulegla awarii!');
AssertFalse(Condition := Executor_Unhappy.Done, 
            Message := 'Executor zglosil sukces (Done), pomimo bledu osi Z!');

TEST_FINISHED();
END_METHOD

METHOD Test_Sequence_ExecutesGroovesCorrectly
VAR_INST
    Step : INT := 0;
    RecipeConfig : ST_RecipeBuilder_Config;
    TestConfig   : ST_GantryXYZ_Config;
END_VAR
TEST('Test_Sequence_ExecutesGroovesCorrectly');

// Wywołujemy CyclicLogic w każdym cyklu zadania PLC, aby test asynchroniczny "żył"
Executor.CyclicLogic();

CASE Step OF
    0:
        // 1. ARRANGE - Przygotowanie receptury BorgoWings (4 frezowania)
        RecipeConfig.PanelFrontLength := 1000.0;
        TestRecipe.Config := RecipeConfig;
        TestRecipe.Build(); 
        
        TestConfig.GroovingSpeedXY := 10;
        TestConfig.GroovingSpeedZ := 10;
        TestConfig.RapidSpeedX := 10;
        TestConfig.RapidSpeedY := 10;
        TestConfig.RapidSpeedZ := 10;
        TestConfig.GroovingIdleTime := 0.0; 
        
        MockConfigProvider.Config := TestConfig;

        // 2. DEPENDENCY INJECTION 
        Executor.RecipeBuilder  := TestRecipe;
        Executor.ConfigProvider := MockConfigProvider;
        Executor.AxisX          := MockAxisX;
        Executor.AxisY          := MockAxisY;
        Executor.AxisZ          := MockAxisZ;
        
        Step := 10;
        
    10:
        // 3. ACT - Start maszyny
        Executor.Execute();
        Step := 20;
        
    20:
        // 4. Czekamy na koniec sekwencji frezowania
        // UWAGA: Test zajmie kilka sekund ze względu na T#500MS w kodzie produkcyjnym (krok 74)
        IF Executor.Done THEN
            Step := 30;
        ELSIF Executor.Error THEN
            AssertTrue(FALSE, 'Executor zwrocil Error zamiast Done podczas frezowania!');
            TEST_FINISHED();
        END_IF
        
    30:
        // 5. ASSERT - BorgoWings ma 4 segmenty, każdy ma 5 przejść.
        // Jeśli Done == TRUE, maszyna stanów prawidłowo przeszła cały proces wielokrotnego zjazdu Z.
        AssertTrue(Condition := Executor.Done, 
                   Message := 'Frezowanie nie doszlo do flagi Done');
                   
        TEST_FINISHED();
END_CASE
END_METHOD

METHOD Test_ZeroSegments_FinishesImmediately
VAR_INST
    i : INT;
END_VAR
TEST('Test_ZeroSegments_FinishesImmediately');

// 1. ARRANGE - Arona zwraca 0 segmentów Groove
Executor_Zero.RecipeBuilder  := BuilderArona;
Executor_Zero.ConfigProvider := MockConfigProvider;
Executor_Zero.AxisX          := MockAxisX;
Executor_Zero.AxisY          := MockAxisY;
Executor_Zero.AxisZ          := MockAxisZ;

// 2. ACT
Executor_Zero.Execute();

FOR i := 1 TO 5 DO
    Executor_Zero.CyclicLogic();
END_FOR

// 3. ASSERT
AssertTrue(Condition := Executor_Zero.Done, 
           Message := 'Executor nie zwrocil Done przy 0 frezowan!');
           
TEST_FINISHED();
END_METHOD

END_FUNCTION_BLOCK

// ---- POUs/TESTS/FB_RecipeBuilder_Test.TcPOU
FUNCTION_BLOCK FB_RecipeBuilder_Test EXTENDS TcUnit.FB_TestSuite
VAR
    BuilderArona 		: FB_PTPArona;
    BuilderBorgoFlaps 	: FB_PTPBorgoFlaps;
	BuilderBorgoWings 	: FB_PTPBorgoWings; 
	BuilderCircle 		: FB_NCICircle;
	BuilderRectangle    : FB_PTPRectangle;
    Config  			: ST_RecipeBuilder_Config;
END_VAR

Test_Arona_Calculates_Segments();
Test_BorgoFlaps_Calculates_Segments();
Test_BorgoWings_Calculates_ActualCopies();
Test_BorgoWings_Calculates_Coordinates();
Test_BorgoWings_Calculates_Footprint();
Test_BorgoWings_Calculates_MaxCopies();
Test_BorgoWings_Calculates_Segments();
Test_BoundaryValues_Are_Clamped();
Test_ExecutionRoute_Assignments();
Test_GlobalOffset_Reduces_MaxCopies();

METHOD Test_Arona_Calculates_Segments
VAR
    WasBuilt : BOOL;
END_VAR
TEST('Test_Arona_Calculates_Segments');

// 1. Arrange - podajemy przykładowe dane wejściowe
Config.PanelFrontLength := 1000.0;
Config.PanelHeight := 100.0;
Config.PanelFrontWidth := 500.0;
Config.RailHeightCorrection := 13.0;
BuilderArona.Config := Config;

// 2. Act - odpalamy wydmuszkę
WasBuilt := BuilderArona.Build();

// 3. Assert - Czy w ogóle przepuścił zabezpieczenie?
AssertTrue(Condition := WasBuilt, 
           Message := 'Przepis zwrocil FALSE - brak implementacji!');

// 4. Assert - Sprawdzamy konkretne wartości dla Arony (po 2 z każdego)
AssertEquals_INT(Expected := 2, 
                 Actual := BuilderArona.SegmentsToCutX, 
                 Message := 'Zla liczba ciec X dla profilu Arona');
                 
AssertEquals_INT(Expected := 2, 
                 Actual := BuilderArona.SegmentsToCutY, 
                 Message := 'Zla liczba ciec Y dla profilu Arona');
                 
AssertEquals_INT(Expected := 2, 
                 Actual := BuilderArona.SegmentsToGroove, 
                 Message := 'Zla liczba frezowan dla profilu Arona');

TEST_FINISHED();
END_METHOD

METHOD Test_BorgoFlaps_Calculates_Segments
VAR
    WasBuilt : BOOL;
END_VAR
TEST('Test_BorgoFlaps_Calculates_Segments');

// 1. Arrange - podajemy przykładowe dane wejściowe
Config.PanelFrontLength := 1000.0;
Config.PanelHeight := 100.0;
Config.PanelFrontWidth := 500.0;
Config.RailHeightCorrection := 13.0;
BuilderBorgoFlaps.Config := Config;

// 2. Act - odpalamy wydmuszkę
WasBuilt := BuilderBorgoFlaps.Build();

// 3. Assert - Czy w ogóle przepuścił zabezpieczenie?
AssertTrue(Condition := WasBuilt, 
           Message := 'Przepis zwrocil FALSE - brak implementacji!');

// 4. Assert - Sprawdzamy konkretne wartości dla Arony (po 2 z każdego)
AssertEquals_INT(Expected := 6, 
                 Actual := BuilderBorgoFlaps.SegmentsToCutX, 
                 Message := 'Zla liczba ciec X dla profilu Borgo Flaps');
                 
AssertEquals_INT(Expected := 6, 
                 Actual := BuilderBorgoFlaps.SegmentsToCutY, 
                 Message := 'Zla liczba ciec Y dla profilu Borgo Flaps');
                 
AssertEquals_INT(Expected := 4, 
                 Actual := BuilderBorgoFlaps.SegmentsToGroove, 
                 Message := 'Zla liczba frezowan dla profilu Borgo Flaps');

TEST_FINISHED();
END_METHOD

METHOD Test_BorgoWings_Calculates_ActualCopies
VAR
    WasBuilt : BOOL;
END_VAR
TEST('Test_BorgoWings_Calculates_ActualCopies');

// ARRANGE - Ustawiamy gabaryty (Wiemy z poprzedniego testu, że Max to 4 w X i 2 w Y)
Config.PanelFrontWidth  := 400.0;
Config.PanelFrontLength := 400.0;
Config.PanelHeight      := 100.0;
Config.CuttingOverpass  := 0.0;
Config.GroovingOverpass := 0.0;

// =========================================================================
// SCENARIUSZ 1: Użytkownik chce wpisać za dużo (np. 10 sztuk), FillAll = FALSE
// =========================================================================
Config.FillAll := FALSE;
Config.RequestedCopiesX := 10; // Kosmos, na płycie wejdą tylko 4
Config.RequestedCopiesY := 10; // Kosmos, na płycie wejdą tylko 2
BuilderBorgoWings.Config := Config;

// ACT 1
WasBuilt := BuilderBorgoWings.Build(); 

// ASSERT 1
AssertEquals_DINT(Expected := 2, 
                 Actual := BuilderBorgoWings.ActualCopiesX, 
                 Message := 'Nie obcieto ActualCopiesX do maksimum przy przekroczeniu!');
                 
AssertEquals_DINT(Expected := 4, 
                 Actual := BuilderBorgoWings.ActualCopiesY, 
                 Message := 'Nie obcieto ActualCopiesY do maksimum przy przekroczeniu!');

// =========================================================================
// SCENARIUSZ 2: Wypełnij całość (FillAll = TRUE)
// =========================================================================
Config.FillAll := TRUE;
Config.RequestedCopiesX := 1; // Operator zostawił 1, ale kliknął "Wypełnij"
Config.RequestedCopiesY := 1;
BuilderBorgoWings.Config := Config;

// ACT 2
WasBuilt := BuilderBorgoWings.Build();

// ASSERT 2
AssertEquals_DINT(Expected := 2, 
                 Actual := BuilderBorgoWings.ActualCopiesX, 
                 Message := 'FillAll=TRUE nie ustawilo ActualCopiesX na Max!');
                 
AssertEquals_DINT(Expected := 4, 
                 Actual := BuilderBorgoWings.ActualCopiesY, 
                 Message := 'FillAll=TRUE nie ustawilo ActualCopiesY na Max!');

TEST_FINISHED();
END_METHOD

METHOD Test_BorgoWings_Calculates_Coordinates
VAR
    WasBuilt : BOOL;
END_VAR


TEST('Test_BorgoWings_Calculates_Coordinates');

// 1. Arrange - wprowadzamy dane
Config.PanelFrontLength := 1000.0;
Config.PanelHeight := 100.0;
Config.PanelFrontWidth := 500.0;
Config.RailHeightCorrection := 13.0;
Config.CuttingOverpass := 20.0;
BuilderBorgoWings.Config := Config;



// 2. Act - budujemy
WasBuilt := BuilderBorgoWings.Build();

AssertTrue(WasBuilt, 'Builder zwrocil FALSE');

// ==========================================
// 3. Assert - SEGMENT CUT X [1] (Zwykłe cięcie)
// ==========================================
AssertEquals_REAL(Expected := 720.0, // TotalX + 20
                  Actual := BuilderBorgoWings.SegmentsCutX[1].Start.X, Delta := 0.01, Message := 'Zly punkt Start.X dla SegmentsCutX[1]');
AssertEquals_REAL(Expected := 600.0, // ShorterX
                  Actual := BuilderBorgoWings.SegmentsCutX[1].Stop.X,  Delta := 0.01, Message := 'Zly punkt Stop.X dla SegmentsCutX[1]');
AssertEquals_REAL(Expected := 1100.0, // ShorterY
                  Actual := BuilderBorgoWings.SegmentsCutX[1].Start.Y, Delta := 0.01, Message := 'Zly punkt Start.Y dla SegmentsCutX[1]');
AssertEquals_REAL(Expected := 1100.0, // ShorterY
                  Actual := BuilderBorgoWings.SegmentsCutX[1].Stop.Y,  Delta := 0.01, Message := 'Zly punkt Stop.Y dla SegmentsCutX[1]');

// ==========================================
// 4. Assert - SEGMENT CUT X [5] i [6] (Korekta o RailHeightCorrection = 13.0)
// ==========================================
// Start.Y dla segmentu 5 to (TotalY - RailHeightCorrection) -> 1200 - 13 = 1187.0
AssertEquals_REAL(Expected := 1187.0, 
                  Actual := BuilderBorgoWings.SegmentsCutX[5].Start.Y, Delta := 0.01, Message := 'Zly punkt Start.Y dla SegmentsCutX[5] (Rail correction)');
// Stop.X dla segmentu 5 to (-CuttingOverpass) -> -20.0
AssertEquals_REAL(Expected := -20.0, 
                  Actual := BuilderBorgoWings.SegmentsCutX[5].Stop.X, Delta := 0.01, Message := 'Zly punkt Stop.X dla SegmentsCutX[5]');

// Start.Y dla segmentu 6 to po prostu RailHeightCorrection -> 13.0
AssertEquals_REAL(Expected := 13.0, 
                  Actual := BuilderBorgoWings.SegmentsCutX[6].Start.Y, Delta := 0.01, Message := 'Zly punkt Start.Y dla SegmentsCutX[6] (Rail correction)');

// ==========================================
// 5. Assert - SEGMENT CUT Y [1] i [5]
// ==========================================
// Segment 1 - Start.Y to (TotalY + CuttingOverpass) -> 1200 + 20 = 1220.0
AssertEquals_REAL(Expected := 1220.0, 
                  Actual := BuilderBorgoWings.SegmentsCutY[1].Start.Y, Delta := 0.01, Message := 'Zly punkt Start.Y dla SegmentsCutY[1]');
// Segment 1 - Start.X to ShorterX -> 600.0
AssertEquals_REAL(Expected := 600.0, 
                  Actual := BuilderBorgoWings.SegmentsCutY[1].Start.X, Delta := 0.01, Message := 'Zly punkt Start.X dla SegmentsCutY[1]');

// Segment 5 - Stop.Y to (-CuttingOverpass) -> -20.0
AssertEquals_REAL(Expected := -20.0, 
                  Actual := BuilderBorgoWings.SegmentsCutY[5].Stop.Y, Delta := 0.01, Message := 'Zly punkt Stop.Y dla SegmentsCutY[5]');
// Segment 5 - Start.X to TotalX -> 700.0
AssertEquals_REAL(Expected := 700.0, 
                  Actual := BuilderBorgoWings.SegmentsCutY[5].Start.X, Delta := 0.01, Message := 'Zly punkt Start.X dla SegmentsCutY[5]');

// ==========================================
// 6. Assert - SEGMENT GROOVE [1]
// ==========================================
// Start.X to TotalX -> 700.0
AssertEquals_REAL(Expected := 700.0, 
                  Actual := BuilderBorgoWings.SegmentsGroove[1].Start.X, Delta := 0.01, Message := 'Zly punkt Start.X dla SegmentsGroove[1]');
// Stop.X to 0
AssertEquals_REAL(Expected := 0.0, 
                  Actual := BuilderBorgoWings.SegmentsGroove[1].Stop.X, Delta := 0.01, Message := 'Zly punkt Stop.X dla SegmentsGroove[1]');

TEST_FINISHED();
END_METHOD

METHOD Test_BorgoWings_Calculates_Footprint
VAR
    WasBuilt : BOOL;
END_VAR
TEST('Test_BorgoWings_Calculates_Footprint');

// 1. Arrange - Wymiary z Twojego HMI
Config.PanelFrontWidth  := 400.0;
Config.PanelFrontLength := 400.0;
Config.PanelHeight      := 100.0;
Config.CuttingOverpass  := 0.0;
Config.GroovingOverpass := 0.0;

BuilderBorgoWings.Config := Config;

// 2. Act
WasBuilt := BuilderBorgoWings.Build();

// 3. Assert - Całkowity wymiar cięcia na płycie
// TotalX = PanelFrontWidth (400) + 2 * PanelHeight (200) = 600.0
AssertEquals_REAL(Expected := 600.0, 
                  Actual := BuilderBorgoWings.FootprintX, 
                  Delta := 0.01, 
                  Message := 'Zle wyliczony gabaryt X (FootprintX) dla BorgoWings!');

// TotalY = PanelFrontLength (400) + 2 * PanelHeight (200) = 600.0
AssertEquals_REAL(Expected := 600.0, 
                  Actual := BuilderBorgoWings.FootprintY, 
                  Delta := 0.01, 
                  Message := 'Zle wyliczony gabaryt Y (FootprintY) dla BorgoWings!');

TEST_FINISHED();
END_METHOD

METHOD Test_BorgoWings_Calculates_MaxCopies
VAR
    WasBuilt : BOOL;
END_VAR
TEST('Test_BorgoWings_Calculates_MaxCopies');

// 1. Arrange
Config.PanelFrontWidth  := 400.0;
Config.PanelFrontLength := 400.0;
Config.PanelHeight      := 100.0;
Config.CuttingOverpass  := 0.0;
Config.GroovingOverpass := 0.0;
BuilderBorgoWings.Config := Config;

// 2. Act
WasBuilt := BuilderBorgoWings.Build();

// 3. Assert
AssertEquals_DINT(Expected := 2, 
                 Actual := BuilderBorgoWings.MaxCopiesX, 
                 Message := 'Zle wyliczona maksymalna liczba sztuk w osi X!');


AssertEquals_DINT(Expected := 4, 
                 Actual := BuilderBorgoWings.MaxCopiesY, 
                 Message := 'Zle wyliczona maksymalna liczba sztuk w osi Y!');

TEST_FINISHED();
END_METHOD

METHOD Test_BorgoWings_Calculates_Segments
VAR
    WasBuilt : BOOL;
END_VAR
TEST('Test_BorgoWings_Calculates_Segments');

// 1. Arrange - podajemy przykładowe dane wejściowe
Config.PanelFrontLength := 1000.0;
Config.PanelHeight := 100.0;
Config.PanelFrontWidth := 500.0;
Config.RailHeightCorrection := 13.0;
BuilderBorgoWings.Config := Config;

// 2. Act - odpalamy wydmuszkę
WasBuilt := BuilderBorgoWings.Build();

// 3. Assert - Czy w ogóle przepuścił zabezpieczenie?
AssertTrue(Condition := WasBuilt, 
           Message := 'Przepis zwrocil FALSE - brak implementacji!');

// 4. Assert - Sprawdzamy konkretne wartości dla Arony (po 2 z każdego)
AssertEquals_INT(Expected := 6, 
                 Actual := BuilderBorgoWings.SegmentsToCutX, 
                 Message := 'Zla liczba ciec X dla profilu Borgo Wings');
                 
AssertEquals_INT(Expected := 6, 
                 Actual := BuilderBorgoWings.SegmentsToCutY, 
                 Message := 'Zla liczba ciec Y dla profilu Borgo Wings');
                 
AssertEquals_INT(Expected := 4, 
                 Actual := BuilderBorgoWings.SegmentsToGroove, 
                 Message := 'Zla liczba frezowan dla profilu Borgo Wings');

TEST_FINISHED();
END_METHOD

METHOD Test_BoundaryValues_Are_Clamped
VAR
    TestConfig : ST_RecipeBuilder_Config;
    ActualConfig : ST_RecipeBuilder_Config;
END_VAR
TEST('Test_BoundaryValues_Are_Clamped');

// 1. ARRANGE - Ekstremalnie złe wartości z "HMI"
TestConfig.PanelFrontLength := -500.0;     // Ujemna długość!
TestConfig.PanelFrontWidth  := 999999.0;   // Kosmiczna szerokość!
TestConfig.PanelHeight      := 0.0;        // Zerowa wysokość (grozi dzieleniem przez 0!)

// 2. ACT - Próba wstrzyknięcia złych danych do Buildera
BuilderBorgoWings.Config := TestConfig; 
ActualConfig := BuilderBorgoWings.Config; // Odczytujemy to, co Builder fizycznie zapisał

// 3. ASSERT - Sprawdzamy czy Builder użył funkcji LIMIT
AssertEquals_REAL(Expected := 100.0, // Założone minimum dla długości
                  Actual := ActualConfig.PanelFrontLength, 
                  Delta := 0.01, 
                  Message := 'Ujemna dlugosc nie zostala przycieta do minimum!');

AssertEquals_REAL(Expected := 1234.0, // Założone maximum dla szerokości z Twojego HMI
                  Actual := ActualConfig.PanelFrontWidth, 
                  Delta := 0.01, 
                  Message := 'Kosmiczna szerokosc nie zostala przycieta do maximum!');

AssertEquals_REAL(Expected := 0.0, // Założone minimum dla wysokości z Twojego HMI
                  Actual := ActualConfig.PanelHeight, 
                  Delta := 0.01, 
                  Message := 'Zerowa wysokosc nie zostala bezpiecznie ograniczona!');

TEST_FINISHED();
END_METHOD

METHOD Test_ExecutionRoute_Assignments
VAR_INST
END_VAR
TEST('Test_ExecutionRoute_Assignments');

// ASSERT - Sprawdzamy czy każdy z builderów prawidłowo zgłasza swój format do maszyny stanów Gantry
AssertEquals_INT(Expected := E_ExecutionRoute.ePTP, 
                 Actual := BuilderArona.ExecutionRoute, 
                 Message := 'Arona powinna byc obslugiwana przez ścieżkę ePTP');
                 
AssertEquals_INT(Expected := E_ExecutionRoute.ePTP, 
                 Actual := BuilderBorgoFlaps.ExecutionRoute, 
                 Message := 'BorgoFlaps powinna byc obslugiwana przez ścieżkę ePTP');
                 
AssertEquals_INT(Expected := E_ExecutionRoute.ePTP, 
                 Actual := BuilderBorgoWings.ExecutionRoute, 
                 Message := 'BorgoWings powinna byc obslugiwana przez ścieżkę ePTP');
                 
AssertEquals_INT(Expected := E_ExecutionRoute.eGCode, 
                 Actual := BuilderCircle.ExecutionRoute, 
                 Message := 'Circle powinien byc obslugiwany przez ścieżkę eGCode');
                 
AssertEquals_INT(Expected := E_ExecutionRoute.ePTP, 
                 Actual := BuilderRectangle.ExecutionRoute, 
                 Message := 'Rectangle powinien byc obslugiwany przez ścieżkę ePTP');

TEST_FINISHED();
END_METHOD

METHOD Test_GlobalOffset_Reduces_MaxCopies
VAR_INST 
    LocalBuilder       : FB_PTPBorgoWings;
    MockConfigProvider : FB_MockConfigProvider;
END_VAR
VAR 
    MachineConfig      : ST_GantryXYZ_Config;
    TestConfig         : ST_RecipeBuilder_Config;
    WasBuilt           : BOOL;
END_VAR
TEST('Test_GlobalOffset_Reduces_MaxCopies');

// 1. ARRANGE
// Wymiary detalu: Szer=400, Dlug=400, Wys=100.
// Gabaryt roboczy (Footprint) to Nominal + 2*Wysokosc -> 600x600 mm.
TestConfig.PanelFrontWidth  := 400.0;
TestConfig.PanelFrontLength := 400.0;
TestConfig.PanelHeight      := 100.0;
TestConfig.CuttingOverpass  := 0.0;
TestConfig.GroovingOverpass := 0.0;

// Konfiguracja maszyny: "Zjadamy" stół offsetami!
// Surowa plyta ma 1200 x 2400 mm
MachineConfig.RawBoardX := 1200.0; // <--- DODAJ TO
MachineConfig.RawBoardY := 2400.0; // <--- DODAJ TO
MachineConfig.GlobalOffsetX := 300.0;  // Zostaje 900 mm dla osi X
MachineConfig.GlobalOffsetY := 1000.0; // Zostaje 1400 mm dla osi Y
MockConfigProvider.Config := MachineConfig;

// Wstrzykujemy zależności
LocalBuilder.ConfigProvider := MockConfigProvider;
LocalBuilder.Config := TestConfig;

// 2. ACT
WasBuilt := LocalBuilder.Build();

// 3. ASSERT
// Os X: Zostalo 900 mm. Detal zajmuje 600 mm. TRUNC(900/600) = 1 sztuka (zamiast dotychczasowych 2).
AssertEquals_DINT(Expected := 1, 
                  Actual := LocalBuilder.MaxCopiesX, 
                  Message := 'GlobalOffsetX nie zmniejszyl poprawnie limitu MaxCopiesX!');
                 
// Os Y: Zostalo 1400 mm. Detal zajmuje 600 mm. TRUNC(1400/600) = 2 sztuki (zamiast dotychczasowych 4).
AssertEquals_DINT(Expected := 2, 
                  Actual := LocalBuilder.MaxCopiesY, 
                  Message := 'GlobalOffsetY nie zmniejszyl poprawnie limitu MaxCopiesY!');

TEST_FINISHED();
END_METHOD

END_FUNCTION_BLOCK

// ---- POUs/TESTS/FB_RecipeFactory_Test.TcPOU
FUNCTION_BLOCK FB_RecipeFactory_Test EXTENDS TcUnit.FB_TestSuite
VAR
    Factory : FB_RecipeFactory;
    Config  : ST_RecipeBuilder_Config;
END_VAR

Test_InjectsConfigProviderToAllBuilders();
Test_ReturnsCorrectBuilder();
Test_ReturnsZeroOnInvalidID();
Test_UpdatesConfigForAllBuilders();

METHOD Test_InjectsConfigProviderToAllBuilders
VAR_INST
    MockProvider : FB_MockConfigProvider;
END_VAR
VAR
    TestConfig       : ST_RecipeBuilder_Config;
    BuilderWings     : I_RecipeBuilder;
    BuilderFlaps     : I_RecipeBuilder;
    BuilderArona     : I_RecipeBuilder;
    BuilderCircle    : I_RecipeBuilder;
    BuilderRectangle : I_RecipeBuilder;
    
    iMockProvider    : I_GantryConfigProvider;
END_VAR
TEST('Test_InjectsConfigProviderToAllBuilders');

// 1. ARRANGE
// Rzutujemy instancję bloku na interfejs (aby kompilator wiedział, jak je porównywać)
iMockProvider := MockProvider;

// 2. ACT
Factory.InitializeFactory(Config := TestConfig, ConfigProvider := iMockProvider);

// Wyciągamy instancje z fabryki
BuilderWings     := Factory.GetBuilder(E_RecipeID.ePTPBorgoWings);
BuilderFlaps     := Factory.GetBuilder(E_RecipeID.ePTPBorgoFlaps);
BuilderArona     := Factory.GetBuilder(E_RecipeID.ePTPArona);
BuilderCircle    := Factory.GetBuilder(E_RecipeID.eNCICircle);
BuilderRectangle := Factory.GetBuilder(E_RecipeID.ePTPRectangle);

// 3. ASSERT
AssertTrue(Condition := (BuilderWings.ConfigProvider = iMockProvider),
           Message := 'BuilderWings nie otrzymal wstrzyknietego ConfigProvidera!');
AssertTrue(Condition := (BuilderFlaps.ConfigProvider = iMockProvider),
           Message := 'BuilderFlaps nie otrzymal wstrzyknietego ConfigProvidera!');
AssertTrue(Condition := (BuilderArona.ConfigProvider = iMockProvider),
           Message := 'BuilderArona nie otrzymal wstrzyknietego ConfigProvidera!');
AssertTrue(Condition := (BuilderCircle.ConfigProvider = iMockProvider),
           Message := 'BuilderCircle nie otrzymal wstrzyknietego ConfigProvidera!');
AssertTrue(Condition := (BuilderRectangle.ConfigProvider = iMockProvider),
           Message := 'BuilderRectangle nie otrzymal wstrzyknietego ConfigProvidera!');

TEST_FINISHED();
END_METHOD

METHOD Test_ReturnsCorrectBuilder
VAR
    BuilderWings     : I_RecipeBuilder;
    BuilderFlaps     : I_RecipeBuilder;
    BuilderArona     : I_RecipeBuilder;
    BuilderCircle    : I_RecipeBuilder; // Dodane!
    BuilderRectangle : I_RecipeBuilder; // Dodane!
END_VAR
TEST('Test_ReturnsCorrectBuilder');

// 1. ACT - Prosimy fabrykę o wszystkie wspierane przepisy
BuilderWings     := Factory.GetBuilder(E_RecipeID.ePTPBorgoWings);
BuilderFlaps     := Factory.GetBuilder(E_RecipeID.ePTPBorgoFlaps);
BuilderArona     := Factory.GetBuilder(E_RecipeID.ePTPArona);
BuilderCircle    := Factory.GetBuilder(E_RecipeID.eNCICircle);
BuilderRectangle := Factory.GetBuilder(E_RecipeID.ePTPRectangle);

// 2. ASSERT - Sprawdzamy, czy żaden z nich nie jest pusty (0)
AssertTrue(Condition := (BuilderWings <> 0), Message := 'Fabryka zwrocila 0 dla eBorgoWings!');
AssertTrue(Condition := (BuilderFlaps <> 0), Message := 'Fabryka zwrocila 0 dla eBorgoFlaps!');
AssertTrue(Condition := (BuilderArona <> 0), Message := 'Fabryka zwrocila 0 dla eArona!');
AssertTrue(Condition := (BuilderCircle <> 0), Message := 'Fabryka zwrocila 0 dla eCircle!');
AssertTrue(Condition := (BuilderRectangle <> 0), Message := 'Fabryka zwrocila 0 dla eRectangle!');

TEST_FINISHED();
END_METHOD

METHOD Test_ReturnsZeroOnInvalidID
VAR
    ReturnedBuilder : I_RecipeBuilder;
END_VAR


TEST('Test_ReturnsZeroOnInvalidID');

// Act - prosimy o eNone (ekran powitalny, bez wybranego programu)
ReturnedBuilder := Factory.GetBuilder(E_RecipeID.eNone);

// Assert - fabryka musi zwrócić 0
AssertTrue(Condition := (ReturnedBuilder = 0), 
           Message := 'Fabryka zwrocila interfejs zamiast 0 dla eNone!');

TEST_FINISHED();
END_METHOD

METHOD Test_UpdatesConfigForAllBuilders
VAR
    TestConfig : ST_RecipeBuilder_Config;
    
    BuilderWings : I_RecipeBuilder;
    BuilderFlaps : I_RecipeBuilder;
    BuilderArona : I_RecipeBuilder;
    
    // Zmienne pomocnicze, żeby obejść błąd kompilatora (odczyt właściwości)
    ActualConfigWings : ST_RecipeBuilder_Config;
    ActualConfigFlaps : ST_RecipeBuilder_Config;
    ActualConfigArona : ST_RecipeBuilder_Config;
END_VAR
TEST('Test_UpdatesConfigForAllBuilders');

// 1. ARRANGE - Tworzymy unikalną, testową konfigurację
TestConfig.PanelFrontLength := 999.0;
TestConfig.PanelHeight := 111.0;

// 2. ACT - Wrzucamy ją do fabryki, żeby rozesłała dalej
Factory.UpdateConfig(TestConfig);

// 3. Wyciągamy instancje z fabryki
BuilderWings := Factory.GetBuilder(E_RecipeID.ePTPBorgoWings);
BuilderFlaps := Factory.GetBuilder(E_RecipeID.ePTPBorgoFlaps);
BuilderArona := Factory.GetBuilder(E_RecipeID.ePTPArona);

// Zgrywamy konfigurację z właściwości interfejsów do zmiennych lokalnych
ActualConfigWings := BuilderWings.Config;
ActualConfigFlaps := BuilderFlaps.Config;
ActualConfigArona := BuilderArona.Config;

// 4. ASSERT - Sprawdzamy, czy wszyscy mają tę samą wartość
AssertEquals_REAL(Expected := 999.0, 
                  Actual := ActualConfigWings.PanelFrontLength, 
                  Delta := 0.01, 
                  Message := 'BuilderWings nie dostal nowej konfiguracji!');
                  
AssertEquals_REAL(Expected := 999.0, 
                  Actual := ActualConfigFlaps.PanelFrontLength, 
                  Delta := 0.01, 
                  Message := 'BuilderFlaps nie dostal nowej konfiguracji!');
                  
AssertEquals_REAL(Expected := 999.0, 
                  Actual := ActualConfigArona.PanelFrontLength, 
                  Delta := 0.01, 
                  Message := 'BuilderArona nie dostal nowej konfiguracji!');

TEST_FINISHED();
END_METHOD

END_FUNCTION_BLOCK

// ---- POUs/TESTS/FB_Exec_Drill_PTP_Test.TcPOU
FUNCTION_BLOCK FB_Exec_Drill_PTP_Test EXTENDS TcUnit.FB_TestSuite 
VAR
    Executor         : FB_Exec_Drill_PTP;
    Executor_Zero    : FB_Exec_Drill_PTP;
    Executor_Unhappy : FB_Exec_Drill_PTP;
    Executor_Nest    : FB_Exec_Drill_PTP;

    MockConfigProvider : FB_MockConfigProvider;

    MockAxisX     : FB_MockAxis := (Name := 'MockX');
    MockAxisY     : FB_MockAxis := (Name := 'MockY');
    MockAxisZ     : FB_MockAxis := (Name := 'MockZ');
    MockAxisZ_Err : FB_MockAxis := (Name := 'MockZ_Err');
    
    MockRecipe       : FB_MockRecipe_Drill;
    MockRecipe_Zero  : FB_MockRecipe_Drill;
    MockRecipe_Nest  : FB_MockRecipe_Drill;
END_VAR

Test_ZeroHoles_FinishesImmediately();
Test_AxisError_AbortsSequence();
Test_Sequence_ExecutesDrillCorrectly();
Test_Sequence_ExecutesNestingCorrectly();

METHOD Test_AxisError_AbortsSequence
VAR_INST
    i : INT;
    TestConfig : ST_GantryXYZ_Config;
END_VAR
TEST('Test_AxisError_AbortsSequence');

// 1. ARRANGE - Używamy receptury z 2 otworami
MockRecipe.TestHolesCount := 2;        
MockRecipe.Build();                       

MockConfigProvider.Config := TestConfig;

Executor_Unhappy.RecipeBuilder  := MockRecipe;
Executor_Unhappy.ConfigProvider := MockConfigProvider;
Executor_Unhappy.AxisX          := MockAxisX;
Executor_Unhappy.AxisY          := MockAxisY;
Executor_Unhappy.AxisZ          := MockAxisZ_Err; // Oś ulegnie awarii!

MockAxisZ_Err.ForceError := TRUE;

// 2. ACT
Executor_Unhappy.Execute();

// Puszczamy maszynę stanów na kilka cykli 
FOR i := 1 TO 10 DO
    Executor_Unhappy.CyclicLogic();
END_FOR

// 3. ASSERT
AssertTrue(Condition := Executor_Unhappy.Error, 
           Message := 'Executor nie zglosil bledu, gdy os Z (wiertlo) ulegla awarii!');
AssertFalse(Condition := Executor_Unhappy.Done, 
            Message := 'Executor zglosil sukces (Done), pomimo bledu osi!');

TEST_FINISHED();
END_METHOD

METHOD Test_Sequence_ExecutesDrillCorrectly
VAR_INST
    Step : INT := 0;
    TestConfig : ST_GantryXYZ_Config;
END_VAR
TEST('Test_Sequence_ExecutesDrillCorrectly');
Executor.CyclicLogic();

CASE Step OF
    0:
        // 1. ARRANGE
        MockRecipe.TestHolesCount := 2;
        MockRecipe.Build(); 
        
        TestConfig.GroovingSpeedZ := 10;
        TestConfig.RapidSpeedX := 10;
        TestConfig.RapidSpeedY := 10;
        TestConfig.RapidSpeedZ := 10;
        TestConfig.GroovingIdleTime := 0.0; // Ucinamy czas oczekiwania, żeby test był natychmiastowy!
        
        MockConfigProvider.Config := TestConfig;

        Executor.RecipeBuilder  := MockRecipe;
        Executor.ConfigProvider := MockConfigProvider;
        Executor.AxisX          := MockAxisX;
        Executor.AxisY          := MockAxisY;
        Executor.AxisZ          := MockAxisZ;
        
        Step := 10;

    10:
        // 2. ACT
        Executor.Execute();
        Step := 20;
        
    20:
        // 3. Czekamy na koniec asynchronicznej sekwencji wiercenia
        IF Executor.Done THEN
            Step := 30;
        ELSIF Executor.Error THEN
            AssertTrue(FALSE, 'Executor zwrocil Error zamiast Done podczas standardowego wiercenia!');
            TEST_FINISHED();
        END_IF
        
    30:
        // 4. ASSERT
        AssertTrue(Condition := Executor.Done, Message := 'Wiercenie nie doszlo do flagi Done');
        TEST_FINISHED();
END_CASE
END_METHOD

METHOD Test_Sequence_ExecutesNestingCorrectly
VAR_INST
    Step : INT := 0;
    TestConfig : ST_GantryXYZ_Config;
END_VAR
TEST('Test_Sequence_ExecutesNestingCorrectly');
Executor_Nest.CyclicLogic();

CASE Step OF
    0:
        // 1. ARRANGE - 2 otwory, ale aż 4 kopie (2x2 na płycie) -> Łącznie do wykonania 8 wierceń
        MockRecipe_Nest.TestHolesCount := 2;
        MockRecipe_Nest.TestCopiesX := 2;
        MockRecipe_Nest.TestCopiesY := 2;
        MockRecipe_Nest.Build(); 
        
        TestConfig.GroovingSpeedZ := 10;
        TestConfig.RapidSpeedX := 10;
        TestConfig.RapidSpeedY := 10;
        TestConfig.RapidSpeedZ := 10;
        TestConfig.GroovingIdleTime := 0.0;
        
        MockConfigProvider.Config := TestConfig;

        Executor_Nest.RecipeBuilder  := MockRecipe_Nest;
        Executor_Nest.ConfigProvider := MockConfigProvider;
        Executor_Nest.AxisX          := MockAxisX;
        Executor_Nest.AxisY          := MockAxisY;
        Executor_Nest.AxisZ          := MockAxisZ;
        
        Step := 10;

    10:
        // 2. ACT
        Executor_Nest.Execute();
        Step := 20;
        
    20:
        IF Executor_Nest.Done THEN
            Step := 30;
        ELSIF Executor_Nest.Error THEN
            AssertTrue(FALSE, 'Executor zwrocil Error podczas Nestingu!');
            TEST_FINISHED();
        END_IF
        
    30:
        // 3. ASSERT
        AssertTrue(Condition := Executor_Nest.Done, Message := 'Wiercenie (Nesting) nie doszlo do flagi Done');
        TEST_FINISHED();
END_CASE
END_METHOD

METHOD Test_ZeroHoles_FinishesImmediately
VAR_INST
    i : INT;
END_VAR
TEST('Test_ZeroHoles_FinishesImmediately');

// 1. ARRANGE - Udajemy, że nie ma otworów do zrobienia (częsty przypadek dla wielu części)
MockRecipe_Zero.TestHolesCount := 0;
MockRecipe_Zero.Build();

Executor_Zero.RecipeBuilder  := MockRecipe_Zero;
Executor_Zero.ConfigProvider := MockConfigProvider;
Executor_Zero.AxisX          := MockAxisX;
Executor_Zero.AxisY          := MockAxisY;
Executor_Zero.AxisZ          := MockAxisZ;

// 2. ACT
Executor_Zero.Execute();

// Zgodnie z kodem, przy <= 0 otworów, maszyna przechodzi z 5 od razu na 1000 i zamyka zadanie. Puszczamy na kilka cykli.
FOR i := 1 TO 5 DO
    Executor_Zero.CyclicLogic();
END_FOR

// 3. ASSERT
AssertTrue(Condition := Executor_Zero.Done, 
           Message := 'Executor nie zwrocil Done przy 0 otworow do wywiercenia!');

TEST_FINISHED();
END_METHOD

END_FUNCTION_BLOCK

// ---- POUs/TESTS/Mocks/FB_MockRecipe_Drill.TcPOU
FUNCTION_BLOCK FB_MockRecipe_Drill EXTENDS FB_RecipeBase
VAR_INPUT
    TestHolesCount : INT := 2;
    TestCopiesX    : DINT := 1;
    TestCopiesY    : DINT := 1;
END_VAR

METHOD Build : BOOL
// Ustawiamy wymiary wirtualnej płyty i limity
_NominalX := 1000.0;
_NominalY := 1000.0;

_Config.IsValid := TRUE;

// Wstrzykujemy zadane w teście wartości ilości otworów
_HolesToDrill := TestHolesCount;

// Sztuczne współrzędne dla max 4 otworów
IF TestHolesCount >= 1 THEN _HolesDrill[1].X := 10.0; _HolesDrill[1].Y := 10.0; END_IF
IF TestHolesCount >= 2 THEN _HolesDrill[2].X := 20.0; _HolesDrill[2].Y := 20.0; END_IF
IF TestHolesCount >= 3 THEN _HolesDrill[3].X := 30.0; _HolesDrill[3].Y := 30.0; END_IF
IF TestHolesCount >= 4 THEN _HolesDrill[4].X := 40.0; _HolesDrill[4].Y := 40.0; END_IF

// Symulacja wyliczonego Nestingu (ilości sztuk)
_ActualCopiesX := TestCopiesX;
_ActualCopiesY := TestCopiesY;

_Done := TRUE;
_Busy := FALSE;
Build := TRUE;
END_METHOD

END_FUNCTION_BLOCK

// ---- POUs/GlobalTextList.TcGTLO
TEXTLIST GlobalTextList
  150 = ' %s'
  816 = '%0.2f'
  380 = '%0.2f%%'
  685 = '%s'
  53 = '+X'
  797 = '+Y'
  325 = '+Z'
  93 = '-X'
  174 = '-Y'
  670 = '-Z'
  296 = '40'
  525 = 'Arona'
  758 = 'Back'
  845 = 'Before Start'
  847 = 'Before Start Choose Your Program'
  992 = 'Borgo Flaps'
  573 = 'Borgo Wings'
  643 = 'Choose Parameters'
  501 = 'Choose Program'
  416 = 'Choose program'
  385 = 'Choose Program ->'
  163 = 'Clean'
  452 = 'Clear'
  233 = 'Cooling'
  820 = 'Copies X'
  104 = 'Copies X\\'
  567 = 'Copies Y'
  810 = 'Current Speed'
  836 = 'Cutter X Offset X'
  817 = 'Cutter X Offset Y'
  943 = 'Cutter Y Offset X'
  49 = 'Cutter Y OFfset Y'
  123 = 'Cutter Y Offset Y'
  108 = 'Cutting Heigt Z'
  47 = 'Cutting Idle Time'
  177 = 'Cutting Speed X'
  638 = 'Cutting Speed x'
  942 = 'Cutting Speed XY'
  270 = 'Cutting Speed Y'
  372 = 'Cutting Speed Z'
  119 = 'Cutting Tool Overpass'
  194 = 'Diameter'
  925 = 'Dimension correction'
  853 = 'Fill All'
  796 = 'Global Offset'
  610 = 'Global Offset X'
  201 = 'Global Offset Y'
  220 = 'Global Offset Z'
  340 = 'Global OffsetX'
  245 = 'GlobalOffset'
  363 = 'Groove Depth'
  524 = 'Grooving Height'
  539 = 'Grooving Idle Time'
  373 = 'Grooving Speed X'
  27 = 'Grooving Speed XY'
  263 = 'Grooving Speed Y'
  55 = 'Grooving Speed Z'
  188 = 'Grooving Tool Overpass'
  600 = 'Happy Cutting :)'
  719 = 'Happy Cutting:)'
  241 = 'HMI_GantryXYZ.Co'
  557 = 'Idle Time'
  208 = 'Info'
  999 = 'Label'
  564 = 'Length'
  18 = 'Leveling'
  46 = 'Maintenance'
  655 = 'Maintenance Mode'
  904 = 'Manual'
  890 = 'Manual Mode'
  67 = 'Not Implemented'
  371 = 'Override'
  537 = 'PackML State'
  203 = 'Panel Front Length'
  415 = 'Panel Front Width'
  565 = 'Panel Height'
  512 = 'Panel Length'
  337 = 'Panel Width'
  369 = 'Panels'
  914 = 'Parameters'
  115 = 'PRODCTION'
  929 = 'Production'
  289 = 'PRODUCTION'
  749 = 'PRODUCTION IN PROGRESS'
  453 = 'Production Mode'
  94 = 'Program %'
  218 = 'Program Set: %s'
  412 = 'Program: %s'
  779 = 'Progress'
  209 = 'Radius'
  876 = 'Rail Height'
  883 = 'Rail Height Correction'
  1109 = 'Rapid Speed Q'
  393 = 'Rapid Speed X'
  930 = 'Rapid Speed Y'
  939 = 'Rapid Speed Z'
  744 = 'RawBoardX'
  334 = 'RawBoardY'
  646 = 'RawBoardZ'
  302 = 'Reboot Machine'
  181 = 'Reset'
  271 = 'Safe Clearance Z'
  526 = 'Set Z Offset'
  513 = 'Spindle'
  0 = 'Spindle Offset X'
  644 = 'Spindle Offset Y'
  740 = 'Start'
  77 = 'START'
  701 = 'Start Arona'
  915 = 'Start Borgo Flaps'
  483 = 'Start Borgo Wings'
  516 = 'State: %s'
  618 = 'Step %'
  98 = 'STOP'
  851 = 'Tool Overpass'
  294 = 'Tool Override'
  454 = 'Vacuuming'
  76 = 'Vacuuming (not implemented)'
  517 = 'Waiting Time'
  22 = 'Width'
  217 = 'x'
  578 = 'Z Offset'
  677 = 'Zero'
END_TEXTLIST

// ---- VISUs/Modes/ProductionMode/V_Builders.TcVIS
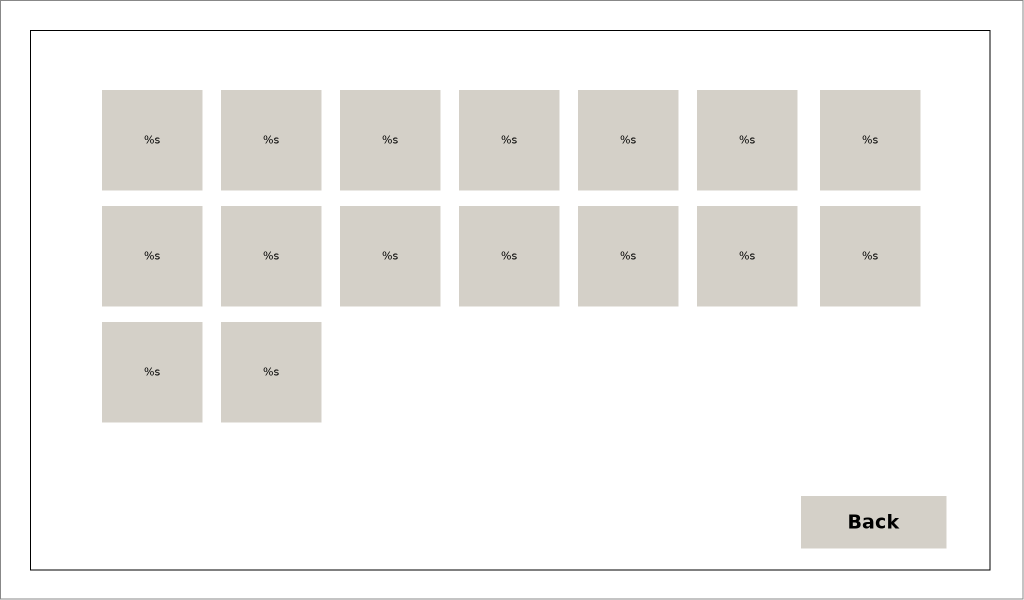
VISUALIZATION V_Builders  // 1024x600
VAR_IN_OUT
	HMI : ST_PackMLBaseModule_HMI;
	HMI_GantryXYZ : ST_GantryXYZ_HMI;
END_VAR
    RoundedRectangle (30,30 960x540)
    RoundedRectangle (801,496 145x52), "Back"
        OnMouseUp: execute { GVL_HMI.PopupToDisplay := 0; }
    RoundedRectangle (340,90 100x100), "%s", text variable: MAIN.Seedra.aRecipeNames[3], colour toggle: HMI_GantryXYZ.Command.ProgramIdRequested = 3, invisible if: MAIN.Seedra.aRecipeNames[3] = ''
        OnMouseClick: execute { HMI_GantryXYZ.Command.ProgramIdRequested := 3; }
        OnMouseUp: execute { GVL_HMI.PopupToDisplay := 0; }
    RoundedRectangle (221,90 100x100), "%s", text variable: MAIN.Seedra.aRecipeNames[2], colour toggle: HMI_GantryXYZ.Command.ProgramIdRequested = 2, invisible if: MAIN.Seedra.aRecipeNames[2] = ''
        OnMouseClick: execute { HMI_GantryXYZ.Command.ProgramIdRequested := 2; }
        OnMouseUp: execute { GVL_HMI.PopupToDisplay := 0; }
    RoundedRectangle (102,90 100x100), "%s", text variable: MAIN.Seedra.aRecipeNames[1], colour toggle: HMI_GantryXYZ.Command.ProgramIdRequested = 1, invisible if: MAIN.Seedra.aRecipeNames[1] = ''
        OnMouseClick: execute { HMI_GantryXYZ.Command.ProgramIdRequested := 1; }
        OnMouseUp: execute { GVL_HMI.PopupToDisplay := 0; }
    RoundedRectangle (459,90 100x100), "%s", text variable: MAIN.Seedra.aRecipeNames[4], colour toggle: HMI_GantryXYZ.Command.ProgramIdRequested = 4, invisible if: MAIN.Seedra.aRecipeNames[4] = ''
        OnMouseClick: execute { HMI_GantryXYZ.Command.ProgramIdRequested := 4; }
        OnMouseUp: execute { GVL_HMI.PopupToDisplay := 0; }
    RoundedRectangle (578,90 100x100), "%s", text variable: MAIN.Seedra.aRecipeNames[5], colour toggle: HMI_GantryXYZ.Command.ProgramIdRequested = 5, invisible if: MAIN.Seedra.aRecipeNames[5] = ''
        OnMouseClick: execute { HMI_GantryXYZ.Command.ProgramIdRequested := 5; }
        OnMouseUp: execute { GVL_HMI.PopupToDisplay := 0; }
    RoundedRectangle (697,90 100x100), "%s", text variable: MAIN.Seedra.aRecipeNames[6], colour toggle: HMI_GantryXYZ.Command.ProgramIdRequested = 6, invisible if: MAIN.Seedra.aRecipeNames[6] = ''
        OnMouseClick: execute { HMI_GantryXYZ.Command.ProgramIdRequested := 6; }
        OnMouseUp: execute { GVL_HMI.PopupToDisplay := 0; }
    RoundedRectangle (820,90 100x100), "%s", text variable: MAIN.Seedra.aRecipeNames[7], colour toggle: HMI_GantryXYZ.Command.ProgramIdRequested = 7, invisible if: MAIN.Seedra.aRecipeNames[7] = ''
        OnMouseClick: execute { HMI_GantryXYZ.Command.ProgramIdRequested := 7; }
        OnMouseUp: execute { GVL_HMI.PopupToDisplay := 0; }
    RoundedRectangle (102,206 100x100), "%s", text variable: MAIN.Seedra.aRecipeNames[8], colour toggle: HMI_GantryXYZ.Command.ProgramIdRequested = 8, invisible if: MAIN.Seedra.aRecipeNames[8] = ''
        OnMouseClick: execute { HMI_GantryXYZ.Command.ProgramIdRequested := 8; }
        OnMouseUp: execute { GVL_HMI.PopupToDisplay := 0; }
    RoundedRectangle (221,206 100x100), "%s", text variable: MAIN.Seedra.aRecipeNames[9], colour toggle: HMI_GantryXYZ.Command.ProgramIdRequested =9, invisible if: MAIN.Seedra.aRecipeNames[9] = ''
        OnMouseClick: execute { HMI_GantryXYZ.Command.ProgramIdRequested := 9; }
        OnMouseUp: execute { GVL_HMI.PopupToDisplay := 0; }
    RoundedRectangle (340,206 100x100), "%s", text variable: MAIN.Seedra.aRecipeNames[10], colour toggle: HMI_GantryXYZ.Command.ProgramIdRequested = 10, invisible if: MAIN.Seedra.aRecipeNames[10] = ''
        OnMouseClick: execute { HMI_GantryXYZ.Command.ProgramIdRequested := 10; }
        OnMouseUp: execute { GVL_HMI.PopupToDisplay := 0; }
    RoundedRectangle (459,206 100x100), "%s", text variable: MAIN.Seedra.aRecipeNames[11], colour toggle: HMI_GantryXYZ.Command.ProgramIdRequested = 11, invisible if: MAIN.Seedra.aRecipeNames[11] = ''
        OnMouseClick: execute { HMI_GantryXYZ.Command.ProgramIdRequested := 11; }
        OnMouseUp: execute { GVL_HMI.PopupToDisplay := 0; }
    RoundedRectangle (578,206 100x100), "%s", text variable: MAIN.Seedra.aRecipeNames[12], colour toggle: HMI_GantryXYZ.Command.ProgramIdRequested = 12, invisible if: MAIN.Seedra.aRecipeNames[12] = ''
        OnMouseClick: execute { HMI_GantryXYZ.Command.ProgramIdRequested := 12; }
        OnMouseUp: execute { GVL_HMI.PopupToDisplay := 0; }
    RoundedRectangle (697,206 100x100), "%s", text variable: MAIN.Seedra.aRecipeNames[13], colour toggle: HMI_GantryXYZ.Command.ProgramIdRequested = 13, invisible if: MAIN.Seedra.aRecipeNames[13] = ''
        OnMouseClick: execute { HMI_GantryXYZ.Command.ProgramIdRequested := 13; }
        OnMouseUp: execute { GVL_HMI.PopupToDisplay := 0; }
    RoundedRectangle (820,206 100x100), "%s", text variable: MAIN.Seedra.aRecipeNames[14], colour toggle: HMI_GantryXYZ.Command.ProgramIdRequested = 14, invisible if: MAIN.Seedra.aRecipeNames[14] = ''
        OnMouseClick: execute { HMI_GantryXYZ.Command.ProgramIdRequested := 14; }
        OnMouseUp: execute { GVL_HMI.PopupToDisplay := 0; }
    RoundedRectangle (102,322 100x100), "%s", text variable: MAIN.Seedra.aRecipeNames[15], colour toggle: HMI_GantryXYZ.Command.ProgramIdRequested = 15, invisible if: MAIN.Seedra.aRecipeNames[15] = ''
        OnMouseClick: execute { HMI_GantryXYZ.Command.ProgramIdRequested := 15; }
        OnMouseUp: execute { GVL_HMI.PopupToDisplay := 0; }
    RoundedRectangle (221,322 100x100), "%s", text variable: MAIN.Seedra.aRecipeNames[16], colour toggle: HMI_GantryXYZ.Command.ProgramIdRequested = 16, invisible if: MAIN.Seedra.aRecipeNames[16] = ''
        OnMouseClick: execute { HMI_GantryXYZ.Command.ProgramIdRequested := 16; }
        OnMouseUp: execute { GVL_HMI.PopupToDisplay := 0; }
END_VISUALIZATION

// ---- VISUs/Modes/ProductionMode/V_Meina2_Samples.TcVIS
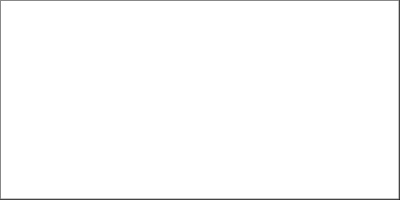
VISUALIZATION V_Meina2_Samples  // 400x200
VAR_IN_OUT
	HMI : ST_PackMLBaseModule_HMI;
	HMI_GantryXYZ : ST_GantryXYZ_HMI;
	HMI_Recipe : ST_RecipeBuilder_HMI;
END_VAR
    RoundedRectangle (0,0 400x200)
END_VISUALIZATION

// ---- VISUs/Modes/ProductionMode/V_ProductionArona.TcVIS
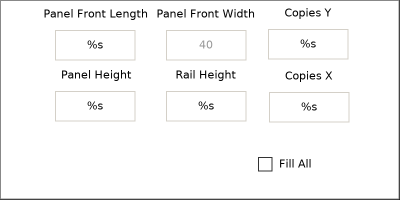
VISUALIZATION V_ProductionArona  // 400x200
VAR_IN_OUT
	HMI : ST_PackMLBaseModule_HMI;
	HMI_GantryXYZ : ST_GantryXYZ_HMI;
	HMI_Recipe : ST_RecipeBuilder_HMI;
END_VAR
    RoundedRectangle (0,0 400x200)
    Textfield (55,30 80x30), "%s", text variable: HMI_Recipe.Config.PanelFrontLength
        OnMouseClick: write the text variable via VisuDialogs.Numpad, min HMI_Recipe.Limits.PanelFrontLength.MinVal, max HMI_Recipe.Limits.PanelFrontLength.MaxVal
    Label (38,4 116x20), "Panel Front Length"
    Textfield (166,30 80x30), "40"
        OnMouseClick: write the text variable via VisuDialogs.Numpad, min HMI_Recipe.Limits.PanelFrontWidth.MinVal, max HMI_Recipe.Limits.PanelFrontWidth.MaxVal
    Label (117,4 178x20), "Panel Front Width"
    Textfield (55,91 80x30), "%s", text variable: HMI_Recipe.Config.PanelHeight
        OnMouseClick: write the text variable via VisuDialogs.Numpad, min HMI_Recipe.Limits.PanelHeight.MinVal, max HMI_Recipe.Limits.PanelHeight.MaxVal
    Label (39,65 115x20), "Panel Height"
    Textfield (166,91 80x30), "%s", text variable: HMI_Recipe.Config.RailHeightCorrection
        OnMouseClick: write the text variable via VisuDialogs.Numpad, min HMI_Recipe.Limits.RailHeightCorrection.MinVal, max HMI_Recipe.Limits.RailHeightCorrection.MaxVal
    Label (155,65 102x20), "Rail Height"
    Checkbox (256,149 72x30), "Fill All", variable: HMI_Recipe.Config.FillAll
    Textfield (269,92 80x30), "%s", text variable: HMI_Recipe.Config.RequestedCopiesX, input disabled if: MAIN.Seedra.RecipeConfig_HMI.Config.FillAll
        OnMouseClick: write the text variable via VisuDialogs.Numpad, min 1, max MAIN.Seedra.RecipeConfig_HMI.Limits.RequestedCopiesX.MaxVal
    Label (258,66 102x20), "Copies X"
    Textfield (268,29 80x30), "%s", text variable: HMI_Recipe.Config.RequestedCopiesY, input disabled if: MAIN.Seedra.RecipeConfig_HMI.Config.FillAll
        OnMouseClick: write the text variable via VisuDialogs.Numpad, min 1, max MAIN.Seedra.RecipeConfig_HMI.Limits.RequestedCopiesY.MaxVal
    Label (257,3 102x20), "Copies Y"
END_VISUALIZATION

// ---- VISUs/Modes/ProductionMode/V_ProductionFeedCircle.TcVIS
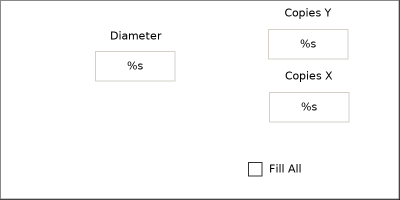
VISUALIZATION V_ProductionFeedCircle  // 400x200
VAR_IN_OUT
	HMI : ST_PackMLBaseModule_HMI;
	HMI_GantryXYZ : ST_GantryXYZ_HMI;
	HMI_Recipe : ST_RecipeBuilder_HMI;
END_VAR
    RoundedRectangle (0,0 400x200)
    Textfield (95,51 80x30), "%s", text variable: HMI_Recipe.Config.Diameter
        OnMouseClick: write the text variable via VisuDialogs.Numpad, min HMI_Recipe.Limits.Diameter.MinVal, max HMI_Recipe.Limits.Diameter.MaxVal
    Label (78,26 116x20), "Diameter"
    Checkbox (246,154 72x30), "Fill All", variable: HMI_Recipe.Config.FillAll
    Textfield (269,92 80x30), "%s", text variable: HMI_Recipe.Config.RequestedCopiesX, input disabled if: MAIN.Seedra.RecipeConfig_HMI.Config.FillAll
        OnMouseClick: write the text variable via VisuDialogs.Numpad, min 1, max MAIN.Seedra.RecipeConfig_HMI.Limits.RequestedCopiesX.MaxVal
    Label (258,66 102x20), "Copies X"
    Textfield (268,29 80x30), "%s", text variable: HMI_Recipe.Config.RequestedCopiesY, input disabled if: MAIN.Seedra.RecipeConfig_HMI.Config.FillAll
        OnMouseClick: write the text variable via VisuDialogs.Numpad, min 1, max MAIN.Seedra.RecipeConfig_HMI.Limits.RequestedCopiesY.MaxVal
    Label (257,3 102x20), "Copies Y"
END_VISUALIZATION

// ---- VISUs/Modes/ProductionMode/V_ProductionMeina2_5Squares.TcVIS
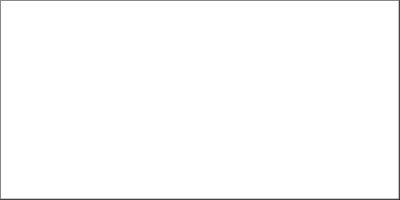
VISUALIZATION V_ProductionMeina2_5Squares  // 400x200
VAR_IN_OUT
	HMI : ST_PackMLBaseModule_HMI;
	HMI_GantryXYZ : ST_GantryXYZ_HMI;
	HMI_Recipe : ST_RecipeBuilder_HMI;
END_VAR
    RoundedRectangle (0,0 400x200)
END_VISUALIZATION

// ---- VISUs/Modes/ProductionMode/V_ProductionMeina2_5Circles.TcVIS
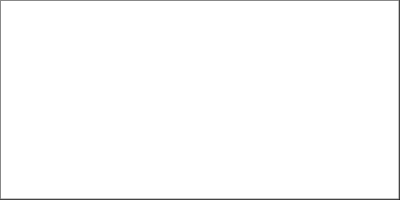
VISUALIZATION V_ProductionMeina2_5Circles  // 400x200
VAR_IN_OUT
	HMI : ST_PackMLBaseModule_HMI;
	HMI_GantryXYZ : ST_GantryXYZ_HMI;
	HMI_Recipe : ST_RecipeBuilder_HMI;
END_VAR
    RoundedRectangle (0,0 400x200)
END_VISUALIZATION

// ---- VISUs/Modes/ProductionMode/V_ProductionMeina2_3Squares.TcVIS
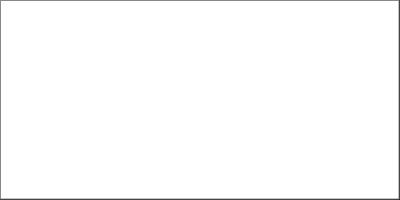
VISUALIZATION V_ProductionMeina2_3Squares  // 400x200
VAR_IN_OUT
	HMI : ST_PackMLBaseModule_HMI;
	HMI_GantryXYZ : ST_GantryXYZ_HMI;
	HMI_Recipe : ST_RecipeBuilder_HMI;
END_VAR
    RoundedRectangle (0,0 400x200)
END_VISUALIZATION

// ---- VISUs/Modes/ProductionMode/V_ProductionMeina2_3Circles.TcVIS
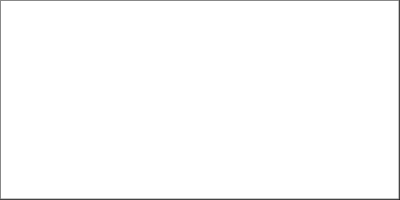
VISUALIZATION V_ProductionMeina2_3Circles  // 400x200
VAR_IN_OUT
	HMI : ST_PackMLBaseModule_HMI;
	HMI_GantryXYZ : ST_GantryXYZ_HMI;
	HMI_Recipe : ST_RecipeBuilder_HMI;
END_VAR
    RoundedRectangle (0,0 400x200)
END_VISUALIZATION

// ---- VISUs/Modes/ProductionMode/V_ProductionMeina2_2Squares.TcVIS
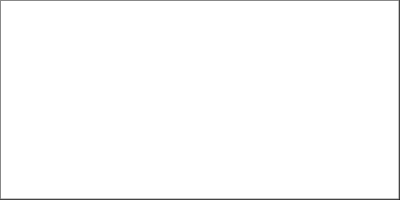
VISUALIZATION V_ProductionMeina2_2Squares  // 400x200
VAR_IN_OUT
	HMI : ST_PackMLBaseModule_HMI;
	HMI_GantryXYZ : ST_GantryXYZ_HMI;
	HMI_Recipe : ST_RecipeBuilder_HMI;
END_VAR
    RoundedRectangle (0,0 400x200)
END_VISUALIZATION

// ---- VISUs/Modes/ProductionMode/V_ProductionMeina2_2Circles.TcVIS
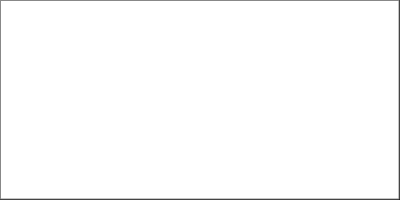
VISUALIZATION V_ProductionMeina2_2Circles  // 400x200
VAR_IN_OUT
	HMI : ST_PackMLBaseModule_HMI;
	HMI_GantryXYZ : ST_GantryXYZ_HMI;
	HMI_Recipe : ST_RecipeBuilder_HMI;
END_VAR
    RoundedRectangle (0,0 400x200)
END_VISUALIZATION

// ---- VISUs/Modes/ProductionMode/V_ProductionMeina2_2Rectangles.TcVIS
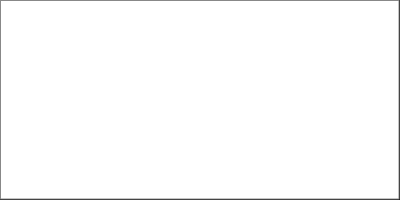
VISUALIZATION V_ProductionMeina2_2Rectangles  // 400x200
VAR_IN_OUT
	HMI : ST_PackMLBaseModule_HMI;
	HMI_GantryXYZ : ST_GantryXYZ_HMI;
	HMI_Recipe : ST_RecipeBuilder_HMI;
END_VAR
    RoundedRectangle (0,0 400x200)
END_VISUALIZATION

// ---- VISUs/Modes/ProductionMode/V_ProductionRoundRectangle.TcVIS
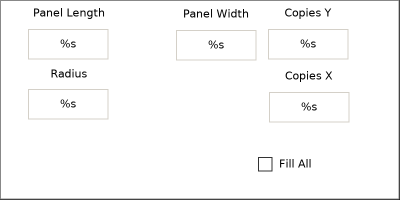
VISUALIZATION V_ProductionRoundRectangle  // 400x200
VAR_IN_OUT
	HMI : ST_PackMLBaseModule_HMI;
	HMI_GantryXYZ : ST_GantryXYZ_HMI;
	HMI_Recipe : ST_RecipeBuilder_HMI;
END_VAR
    RoundedRectangle (0,0 400x200)
    Textfield (28,89 80x30), "%s", text variable: HMI_Recipe.Config.Radius
        OnMouseClick: write the text variable via VisuDialogs.Numpad, min HMI_Recipe.Limits.Radius.MinVal, max HMI_Recipe.Limits.Radius.MaxVal
    Label (11,64 116x20), "Radius"
    Checkbox (256,149 72x30), "Fill All", variable: HMI_Recipe.Config.FillAll
    Textfield (269,92 80x30), "%s", text variable: HMI_Recipe.Config.RequestedCopiesX, input disabled if: MAIN.Seedra.RecipeConfig_HMI.Config.FillAll
        OnMouseClick: write the text variable via VisuDialogs.Numpad, min 1, max MAIN.Seedra.RecipeConfig_HMI.Limits.RequestedCopiesX.MaxVal
    Label (258,66 102x20), "Copies X"
    Textfield (268,29 80x30), "%s", text variable: HMI_Recipe.Config.RequestedCopiesY, input disabled if: MAIN.Seedra.RecipeConfig_HMI.Config.FillAll
        OnMouseClick: write the text variable via VisuDialogs.Numpad, min 1, max MAIN.Seedra.RecipeConfig_HMI.Limits.RequestedCopiesY.MaxVal
    Label (257,3 102x20), "Copies Y"
    Textfield (176,30 80x30), "%s", text variable: HMI_Recipe.Config.PanelFrontWidth
        OnMouseClick: write the text variable via VisuDialogs.Numpad, min HMI_Recipe.Limits.PanelFrontWidth.MinVal, max HMI_Recipe.Limits.PanelFrontWidth.MaxVal
    Textfield (28,29 80x30), "%s", text variable: HMI_Recipe.Config.PanelFrontLength
        OnMouseClick: write the text variable via VisuDialogs.Numpad, min HMI_Recipe.Limits.PanelFrontLength.MinVal, max HMI_Recipe.Limits.PanelFrontLength.MaxVal
    Label (11,3 116x20), "Panel Length"
    Label (127,4 178x20), "Panel Width"
END_VISUALIZATION

// ---- VISUs/Modes/ProductionMode/V_ProductionRectangle.TcVIS
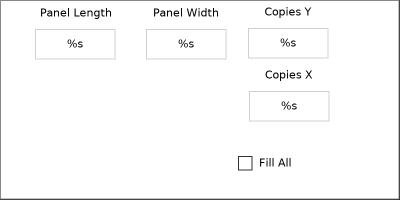
VISUALIZATION V_ProductionRectangle  // 400x200
VAR_IN_OUT
	HMI : ST_PackMLBaseModule_HMI;
	HMI_GantryXYZ : ST_GantryXYZ_HMI;
	HMI_Recipe : ST_RecipeBuilder_HMI;
END_VAR
    RoundedRectangle (0,0 400x200)
    Textfield (35,29 80x30), "%s", text variable: HMI_Recipe.Config.PanelFrontLength
        OnMouseClick: write the text variable via VisuDialogs.Numpad, min HMI_Recipe.Limits.PanelFrontLength.MinVal, max HMI_Recipe.Limits.PanelFrontLength.MaxVal
    Label (18,3 116x20), "Panel Length"
    Textfield (146,29 80x30), "%s", text variable: HMI_Recipe.Config.PanelFrontWidth
        OnMouseClick: write the text variable via VisuDialogs.Numpad, min HMI_Recipe.Limits.PanelFrontWidth.MinVal, max HMI_Recipe.Limits.PanelFrontWidth.MaxVal
    Label (97,3 178x20), "Panel Width"
    Label (135,64 102x20)
    Checkbox (236,148 72x30), "Fill All", variable: HMI_Recipe.Config.FillAll
    Textfield (249,91 80x30), "%s", text variable: HMI_Recipe.Config.RequestedCopiesX, input disabled if: MAIN.Seedra.RecipeConfig_HMI.Config.FillAll
        OnMouseClick: write the text variable via VisuDialogs.Numpad, min 1, max MAIN.Seedra.RecipeConfig_HMI.Limits.RequestedCopiesX.MaxVal
    Label (238,65 102x20), "Copies X"
    Textfield (248,28 80x30), "%s", text variable: HMI_Recipe.Config.RequestedCopiesY, input disabled if: MAIN.Seedra.RecipeConfig_HMI.Config.FillAll
        OnMouseClick: write the text variable via VisuDialogs.Numpad, min 1, max MAIN.Seedra.RecipeConfig_HMI.Limits.RequestedCopiesY.MaxVal
    Label (237,2 102x20), "Copies Y"
END_VISUALIZATION

// ---- VISUs/Modes/ProductionMode/V_ProductionNCICircle.TcVIS
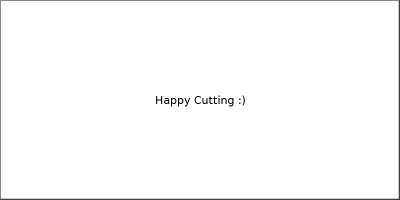
VISUALIZATION V_ProductionNCICircle  // 400x200
VAR_IN_OUT
	HMI : ST_PackMLBaseModule_HMI;
	HMI_GantryXYZ : ST_GantryXYZ_HMI;
	HMI_Recipe : ST_RecipeBuilder_HMI;
END_VAR
    RoundedRectangle (0,0 400x200)
    Label (93,92 215x17), "Happy Cutting :)"
END_VISUALIZATION

